(* CODESYS project CtaAppReport_3.0.0.0.library
   Description: Report Library der CTA
   Version: 3.0.0.0
   Title: CtaAppReport
   Author: SIS
   Company: CTA
   Placeholder: CtaAppReport
   DocFormat: reStructuredText
   CompiledLibraryCompatibilityVersion: CODESYS V3.5 SP16 Patch 3
   LanguageModelAttribute: qualified-access-only
   DefaultNamespace: CtaAppReport

Project tree, tasks and I/O mapping:
  libraries: Standard, 3.5.18.0 (System); CtaAppBmk, 2.0.0.0 (CTA); CtaSysConfig, 1.0.0.2 (CTA); CtaVisSymbols, 1.0.0.0 (CTA); CtaSysEvent, 1.0.0.0 (CTA); VisuDialogs, 3.5.16.20 (System); SysFile, 3.5.17.0 (System); SysDir, 3.5.17.0 (System); VisuSymbols, 4.5.0.0 (System); StringUtils, 3.5.18.0 (System); SysTypes2 Interfaces, * (System); TextListUtils, * (System); CtaAppInfluxLog, 1.0.0.1 (CTA); CtaAppTime, 1.0.0.1 (CTA); SysProcess Implementation, 3.5.17.0 (System); CmpErrors, 3.3.1.40 (System); VisuElemBase, * (System)
  40 Visualizations/
    visualisation REPORT_ID
    TABLE/
      visualisation VIS_REPORT_TABLE
      visualisation VIS_REPORT_TABLE_BASE
      DELETE/
        visualisation VIS_REPORT_DELETE
    PUSHLINE/
      visualisation VIS_REPORT_PUSH_LINE
      visualisation VIS_REPORT_PUSH_LINE_BASE
      visualisation VIS_REPORT_PUSH_LINE_QUERRY
    TABLE LINE/
      visualisation VIS_REPORT_TABLE_LINE_BASE
      visualisation VIS_REPORT_TABLE_LINE_QUERRY
      visualisation VIS_REPORT_TABLE_LINE
    REPORTMANAGER/
      visualisation VIS_REPORTMANAGER
      visualisation VIS_REPORTMANAGER_BASE
    HAND/
      visualisation VIS_REPORT_HAND
    ANZAHL REPORTS/
      visualisation VIS_ANZ_REPORTS_OVERALL
      Modul/
        visualisation VIS_ANZ_REPORTS_MODUL
        visualisation VIS_ANZ_REPORTS_MODUL_BASE
        visualisation VIS_ANZ_REPORTS_MODUL_QUERRY
  30 Program Organization Units/
    CSV/
      function block fbDataHandler [ST]: metWriteDtFrom, FB_INIT, FB_EXIT, actInitPath, proGetCountsOfReports, proExportIdStart, metExportId, metResetCycleCount, proExport, proIsRegistred, metStartDone, metPrepeareStop, proDenyStop, metCyclicCall, metWriteOnChange, metDeleteHistory, metAddObjForeWriteDtFrom, metAddObjForeWriteDtTo, metAddObjForeWriteOnChange
    OBJ/
      function block fbReportObjectFactory [ST]: metQuittAllReports, metDestroyCsvReportObject, metQuittSelectedReports, metCsvGetItf, metDestroyReportObject, metGetItf, metCreateReportObject, proGetNextPos, proGetAktiveReport, proGetActiveErrorMbString, proIsThereAnAktiveError, proGetActiveWarningMbString, metReSaveAfterDelete, metGarbageControll, GetActiveErrorModbusLanguageString
      function block fbReportObject [ST]: proGetReporterText, proGetReportText, proAdditionalText, proCountRetry, proIsQuitt, proIsSelected, proMaxRetry, proReportAcknowledgType, proReportId, proReportTextId, proReportTextList, proReportType, proReporterObjectId, proStateActive, proWritePosInCsv, proQuitt, metSendDataToInflux, metReportObject, proReportIn, proDtFrom, proDtTo, proSetMetaData, metDestroy, proPrio, metWriteDtFromToCsv, metWriteDtToToCsv, metSaveOnChange, metGarbage, GetReportTextLanguage
      function fcWordToHexString [ST]
      function fcReportIdToString8 [ST]
    REPORTER/
      function block fbReportManager [ST]: proWarningText, metSyncReporter, proInfoText, proErrorText, proGetErrorNr, actInit, proGetWarningNr, proGetInfoNr, proAnzError, proAnzWarning, proAnzInfo, proTotalReports
      function block fbReporter [ST]: metGetQuitt, proAktivReport, proHandLokal, proNewReport, metReport, proGetCounts, proDoneReport, proPrio, proOptionalText
    VIS/
      function block fbReportVisu [ST]: metGetReport, metGetShowReport, actConfigFile, proQuittExtern, loadHistory, actEWI, FB_INIT, metReload, FilterWarning, SetFilterId, loadPending, FilterInfo, FilterError, proAnzReportsInTable, proIdMissmatch, MaxOffset
    function fcBmkToId [ST]
    SORT/
      function block fbSort [ST]: metSortPrio, metFilterCustom, proAnzAktiveError, proAnzAktiveInfo, proAnzAktiveReports, proAnzAktiveWarning, proAnzReportsInTable
    program REPORT [ST]
    SQL/
      function Fc_MariaDbDeleteHistory [ST]
      function Fc_MariaDbLogWrite [ST]
      function Fc_MariaDbLogRead [ST]
      function Fc_MariaDbHighestId [ST]
  00000000-0000-0000-0000-000000000000|D:\CoDeSys\LibrariesV3\trunk\Intern\CAA\CAA Template\3.4.0.0 draft\Placeholder.xml
  00000000-0000-0000-0000-000000000000|D:\CoDeSys\LibrariesV3\trunk\Intern\CAA\CAA Template\3.2.0.3 draft\Prefix.pdf
  00000000-0000-0000-0000-000000000000|D:\CoDeSys\LibrariesV3\trunk\Intern\CAA\CAA Template\3.5.2.0 draft\Placeholder.xml
  20 Structs/
    data type enReportType
    data type scPara
    data type scReportMetaData
    data type scReportNr
    data type stReportTextList
    data type enReportacknowledgeType
    data type enTableType
    data type ST_MariaDbLog
  50 Images/
  10 Documenation/
    global variables VersionHistory
    global variables readMe
  21 Interface/
    interface ITF_REPORTMANAGER: proErrorText, proGetWarningNr, metSyncReporter, proGetErrorNr, proGetInfoNr, proInfoText, proWarningText, proTotalReports
    interface ITF_REPORTOBJECT: proGetReportText, proStateActive, proIsQuitt, proIsSelected, proReportId, proMaxRetry, proCountRetry, proReportTextList, proReportTextId, proReporterObjectId, proAdditionalText, proReportType, proReportAcknowledgType, proWritePosInCsv, proGetReporterText, proReportIn, proDtTo, proDtFrom, metReportObject, proQuitt, proSetMetaData, proPrio, metDestroy, metWriteDtFromToCsv, metSaveOnChange, GetReportTextLanguage
  11 Library Parameter/
    global variables Parameter
  12 Konstanten/
    global variables GlobalKonstant
  60 Textlisten/
    text list txtLibAp99_1Error
    text list txtLibAp99_2enTypeOfAck
    text list txtLibAp99_2Warnung
    text list txtLibAp99_3Info
    text list GlobalTextList
    text list txtNoTextList
  13 Globale Variablen/
    global variables GVL_Report
    global variables GVL_REPORT_PERSISTENT
*)

// 20 Structs/enReportType
TYPE enReportType :
(
	Info    := 0,
    Warning := 1,
    Error   := 2
);
END_TYPE

// 20 Structs/scPara
TYPE scPara :
    STRUCT
        fbxEnSafetyFernQuitt            :   CtaSysConfig.fbBOOL;
        fbuiMaxFernQuitt                :   CtaSysConfig.fbUINT;         
    END_STRUCT
END_TYPE

// 20 Structs/scReportMetaData
TYPE scReportMetaData :
    STRUCT
        xReportIn                   :   BOOL;                           // Report Input
        xActive                     :   BOOL;                           // State of Report
        xIsQuitt                    :   BOOL;                           // State of Acknowledge
        xQuitt                      :   BOOL;                           // Acknowledge Flag
        xIsSelected                 :   BOOL;                           // State of Selected in Table
        dtFrom                      :   DT;                             // Date and Time of Report happen
        dtTo                        :   DT;                             // Date and Time of Report gone
        iMaxRetry                   :   INT;                            // Max allowed Retries till Acknowledge is required
        iCountRetry                 :   INT;                            // Retries till now
        stReportTxtId               :   STRING[3];                      // Report Id fore Texlist
        stReportTextList            :   STRING[100];                    // Report TextList 
        uliReportId                 :   ULINT;                          // Report Id build out of BMK and Report Text Id. Ex: Bmk 56M111 & Id 3 = 567711103  
        enReportType                :   enReportType;                   // Type of Report
        enReportacknowledgeType     :   enReportacknowledgeType;        // Type of Report Acknowledge
        stReporterObjId             :   STRING[20];                     // Object Id of Reporter      
        stAdditionalText            :   STRING[20];                     // Additional Text
        dwWritePosInCsv             :   DWORD;                          // Position in Csv File fore write dtTo 
        usiPrio                     :   USINT;                          // Prio
    END_STRUCT
END_TYPE

// 20 Structs/scReportNr
TYPE scReportNr :
    STRUCT
        iError              :   INT;            // Error Status
        usiErrorPrio        :   USINT;
        iWarning            :   INT;            // Warning Status
        usiWarnungPrio      :   USINT;
        iInfo               :   INT;            // Info Status
        usiInfoPrio         :   USINT;
    END_STRUCT
END_TYPE

// 20 Structs/stReportTextList
TYPE stReportTextList : STRING[100]; END_TYPE

// 20 Structs/enReportacknowledgeType
TYPE enReportacknowledgeType :
(
	Auto        := 0,
    Quit        := 1,
    RetryN      := 2
);
END_TYPE

// 20 Structs/enTableType
{attribute 'qualified_only'}
{attribute 'strict'}
TYPE enTableType :
(
	PENDING_REPORTS := 0,
    HISTORY_REPORTS := 1
);
END_TYPE

// 20 Structs/ST_MariaDbLog
TYPE ST_MariaDbLog :
	STRUCT
		id                       : ULINT;
		createdAt                : DT;
		reportType               : enReportType;
		reportId                 : ULINT;
		reporterText             : STRING(150);
		reportText               : STRING(140);
		dtFrom                   : DT;
		dtTo                     : DT;
		isQuitt                  : BOOL;
		reportTextList           : STRING(100);
		reportTextId              : STRING(3);
		reportAcknowledgType     : USINT;
		objectId                 : STRING(20);
		instancePath             : STRING(255);
		additionalText           : STRING(20);
		prio                     : USINT;
		reportIn                  : BOOL;
		stateActive               : BOOL;
	END_STRUCT
END_TYPE

// 10 Documenation/VersionHistory
(* 

.. image:: ../../Images/CTA_Logo.jpg
   :align: right
   :width: 15% 

**Vorlage**   


============ =========== =========== ============================================
**Date**     **Version** **Author**  **Change**
------------ ----------- ----------- --------------------------------------------
04.03.2021   0.0.0.0     SIS         Vorlage erstellt

============ =========== =========== ============================================


*)
VAR_GLOBAL
    stInfo : STRING:= '0.0.0.0, Vorlage, CTA';
END_VAR

// 10 Documenation/readMe
(*

**ReadMe**
 
|	**Empfehlung**
|
|	Die LibAp99aErrorManagement wird benötigt damit aus dem BMK der CTA-E-Schema eine Störungsnummer generiert werden kann. 
|	Es wird für die Ausgabe ein DINT verwendet. Die aufschlüsselung von Buchstaben wird durch die ASCI Nr ersetzt.     
|  
| *Beispiel* 
|
| BMK             =   **56M11**    
| Fehler Nr       =   01-10
| ErrorNr-Modbus  =   BMK    + Fehler Nr
| 56771101        =   567711 + 01
| 56771102        =   567711 + 02
| 56771103        =   567711 + 03
| 56771104        =   567711 + 04
| 56771105        =   567711 + 05
| 56771106        =   567711 + 06
| 56771107        =   567711 + 07 
| 56771108        =   567711 + 08
| 56771109        =   567711 + 09
| 56771110        =   567711 + 10 
|
| Wenn der Fehler keiner BMK zugeordnet werden kann, sollte von der Nr. 1000 hochgezähl werden. 
| Tiefere Nr. werden von den Bibliotheken benötigt. 
*)

VAR_GLOBAL
    xReadMeDone              :   BOOL;
END_VAR

// 13 Globale Variablen/GVL_Report
{attribute 'qualified_only'}
VAR_GLOBAL
    fbReportObjectFactory     :   fbReportObjectFactory;
    fbSort                    :   fbSort;
    fbReportVisu              :   fbReportVisu;
    (* Reports *)             
    ayReportObject            :   ARRAY[1..Parameter.diMaxObject] OF fbReportObject;
    ayItfAktiveReports        :   ARRAY[1..Parameter.diMaxObject] OF ITF_REPORTOBJECT;
    ayItfSortetReportsPrio    :   ARRAY[1..Parameter.diMaxObject] OF ITF_REPORTOBJECT;
    ayItfSortetReportsCustom  :   ARRAY[0..GlobalKonstant.VISU_MAX_NUMBER_OF_CLIENTS] OF ARRAY[1..Parameter.diMaxObject] OF ITF_REPORTOBJECT;
    ayCsvReportObject         :   ARRAY[0..GlobalKonstant.VISU_MAX_NUMBER_OF_CLIENTS] OF ARRAY[0..GlobalKonstant.iUpperSizeTable] OF fbReportObject;
    fbDataHandler             :   fbDataHandler;
    diCountHand               :   DINT;
END_VAR

// 11 Library Parameter/Parameter
{attribute 'qualified_only'}
VAR_GLOBAL CONSTANT
    diMaxObject                  :   DINT :=  150;   // Max 200
    diMaxExportsPerCycle         :   DINT :=  50;    // Kann sich auf die Zykluszeit auswirken wenn zu viele Id pro Zyklus exportiert werden
END_VAR

// 12 Konstanten/GlobalKonstant
{attribute 'qualified_only'}
VAR_GLOBAL CONSTANT
    stTextListWarning           :   stReportTextList    := 'CtaAppReport.txtLibAp99_2Warnung';
    stTextListInfo              :   stReportTextList    := 'CtaAppReport.txtLibAp99_3Info';
    iUpperSizeTable             :   INT                 := 13;   
	VISU_MAX_NUMBER_OF_CLIENTS	:	INT					:= 15;
END_VAR

// 13 Globale Variablen/GVL_REPORT_PERSISTENT
{attribute 'qualified_only'}
VAR_GLOBAL RETAIN 
	scLastErrorReport         :   scReportMetaData;
	scLastWarningReport       :   scReportMetaData;
	scLastInfoReport          :   scReportMetaData;  
END_VAR

// 21 Interface/ITF_REPORTMANAGER
INTERFACE ITF_REPORTMANAGER EXTENDS __SYSTEM.IQueryInterface

PROPERTY proErrorText : STRING[100]
GET
END_GET
END_PROPERTY

PROPERTY proGetWarningNr : INT
GET
END_GET
END_PROPERTY

METHOD metSyncReporter : BOOL
VAR_INPUT
	refFbReporter	:	REFERENCE TO fbReporter;
END_VAR
END_METHOD

PROPERTY proGetErrorNr : INT
GET
END_GET
END_PROPERTY

PROPERTY proGetInfoNr : INT
GET
END_GET
END_PROPERTY

PROPERTY proInfoText : STRING[100]
GET
END_GET
END_PROPERTY

PROPERTY proWarningText : STRING[100]
GET
END_GET
END_PROPERTY

PROPERTY proTotalReports : INT
GET
END_GET
END_PROPERTY

END_INTERFACE

// 30 Program Organization Units/REPORTER/fbReporter
FUNCTION_BLOCK FINAL fbReporter 
VAR
	diArrayReportAdr     :	DINT;
	iCountReports		 :	INT;
	tonDelay			 :	TON;
	tonReset			 :	TON;
	_stReportTextList    :	POINTER TO stReportTextList;
	_iReportID			 :  INT;
	xNewReport			 :  BOOL;
	xAktiveReport		 :  BOOL;
    xDoneReport          :  BOOL;
	_enReportType        :  enReportType;
    xHand                :  BOOL;
    usiPrio              :  USINT;
    xExportDone          :  BOOL; 
    xInitDone            :  BOOL;
END_VAR

METHOD metGetQuitt : BOOL
VAR
    ITF_REPORTOBJECT : ITF_REPORTOBJECT;
END_VAR
IF diArrayReportAdr >= 1 THEN
    IF __QUERYINTERFACE(GVL_Report.fbReportObjectFactory.metGetItf(diArrayReportAdr),ITF_REPORTOBJECT) THEN
        metGetQuitt := ITF_REPORTOBJECT.proIsQuitt;
    END_IF;
ELSE
    metGetQuitt := FALSE;
END_IF
END_METHOD

PROPERTY proAktivReport : BOOL
GET
proAktivReport := xAktiveReport;
END_GET
END_PROPERTY

PROPERTY proHandLokal : BOOL
SET
IF proHandLokal AND  NOT xHand THEN
    GVL_Report.diCountHand := GVL_Report.diCountHand + 1;
    xHand := TRUE;
ELSIF NOT proHandLokal AND xHand THEN
    GVL_Report.diCountHand := GVL_Report.diCountHand - 1;
    IF GVL_Report.diCountHand < 0 THEN
        GVL_Report.diCountHand := 0;
	END_IF;
    xHand := FALSE;    
END_IF;
END_SET
END_PROPERTY

PROPERTY INTERNAL proNewReport : BOOL
SET
xNewReport := proNewReport;
END_SET
GET
proNewReport := xNewReport;
END_GET
END_PROPERTY

METHOD FINAL metReport : BOOL
VAR_INPUT
    xSetReportIn          		:   BOOL;
    iReportID           		:   INT;
    enReportTypeIn      		:   enReportType;
    enReportAcknowledgeTypeIn   :   enReportAcknowledgeType;
	tDelay              		:   TIME;  
	ITF_BMK_IN					:	CtaAppBmk.ITF_BMK;
	pstReportTextListIn 		:	POINTER TO stReportTextList;	 
	stOptionalReportText		:	STRING[20];	
    iRetryTilReportLock 		:   INT;                            
    xResetCount         		:   BOOL;                            
	tReset						:	TIME;                 
END_VAR
VAR
    ITF_REPORTOBJECT            :   ITF_REPORTOBJECT;
END_VAR
IF xInitDone AND_THEN pstReportTextListIn <> 0 AND_THEN ITF_BMK_IN <> 0 THEN
    // Counter mit xResetCount rücksetzen wenn Count < iMaxRetry
    IF tReset > T#0MS AND_THEN enReportAcknowledgeTypeIn = enReportacknowledgeType.RetryN AND_THEN NOT xSetReportIn THEN
        tonReset.IN := iCountReports < iRetryTilReportLock AND iCountReports > 0;
        tonReset.PT	:= tReset;
        tonReset();
	ELSE
		tonReset(IN := FALSE,
				 PT := T#0MS);
    END_IF;
    IF (xResetCount OR tonReset.Q) AND_THEN iCountReports < iRetryTilReportLock AND NOT xSetReportIn  THEN
        diArrayReportAdr := 0;   
        iCountReports := 0;
        tonReset.IN := FALSE;
        tonReset.PT	:= T#0S;	 
        tonReset();
    END_IF;        
	IF xSetReportIn THEN	
		_stReportTextList    := pstReportTextListIn;	
		_iReportID 			 := iReportID;
		_enReportType		 := enReportTypeIn;
	END_IF;
	
	tonDelay.IN          := xSetReportIn;
	tonDelay.PT          := tDelay;
	tonDelay();
	(* Wenn Report nicht registriert Registrierprozess starten *)
    IF diArrayReportAdr = 0 THEN
        // Wenn tonDelay.Q aktiv Registrieren      
        IF tonDelay.Q THEN
            (* Create Report Object *)
            diArrayReportAdr := GVL_Report.fbReportObjectFactory.metCreateReportObject();   
            IF diArrayReportAdr <> 0 THEN 
                IF __QUERYINTERFACE(GVL_Report.fbReportObjectFactory.metGetItf(diArrayReportAdr),ITF_REPORTOBJECT) THEN               
                    (* Set Infos *)  
                    xNewReport := TRUE;
                    xAktiveReport := TRUE;
                    iCountReports := iCountReports + 1;
                    ITF_REPORTOBJECT.proReportType              :=  enReportTypeIn;                         // Report Type
                    ITF_REPORTOBJECT.proReportAcknowledgType    :=  enReportAcknowledgeTypeIn;              // Report Acknowledge Type
                    ITF_REPORTOBJECT.proReportTextId            :=  TO_STRING(iReportID);                   // Report Id
                    ITF_REPORTOBJECT.proReportTextList          :=  pstReportTextListIn^;                   // Report Text list
                    ITF_REPORTOBJECT.proReporterObjectId        :=  ITF_BMK_IN.proGetObjectId;              // Reporter Object Id
                    ITF_REPORTOBJECT.proSetInstancePath         :=  ITF_BMK_IN.proGetInstancePath;          // Reporter Instance Path
                    ITF_REPORTOBJECT.proMaxRetry                :=  iRetryTilReportLock;                    // Max Retries
                    ITF_REPORTOBJECT.proCountRetry              :=  iCountReports;                          // Countet Retries
                    ITF_REPORTOBJECT.proAdditionalText          :=  stOptionalReportText;                   // Additional Text
                    ITF_REPORTOBJECT.proReportIn                :=  xSetReportIn;                           // Report Input
                    ITF_REPORTOBJECT.proPrio                    :=  usiPrio;
                    ITF_REPORTOBJECT.metReportObject();                                                     // Call Object              
                END_IF                                                                 
            END_IF;
        END_IF;
    ELSE
        // Zyklische aktualisierung der Daten nach Registrierung       
        IF __QUERYINTERFACE(GVL_Report.fbReportObjectFactory.metGetItf(diArrayReportAdr),ITF_REPORTOBJECT) THEN
            IF ITF_REPORTOBJECT.proReportIn <> xSetReportIn THEN
                ITF_REPORTOBJECT.proReportIn :=  xSetReportIn;                                   // Report Input
            END_IF;
			// Nach Manuellem Quittieren Counts rücksetzen     
			IF ITF_REPORTOBJECT.proQuitt THEN
				iCountReports := 0;
			END_IF;              
			IF NOT ITF_REPORTOBJECT.proStateActive THEN
                xAktiveReport   := FALSE;   
                xDoneReport     := TRUE;
 
                diArrayReportAdr := 0;  
            END_IF;
            ITF_REPORTOBJECT.metReportObject();                                                             // Call Object 
        ELSE
            diArrayReportAdr := 0;
            xAktiveReport   := FALSE; 
            xDoneReport     := TRUE;
        END_IF;                                              
    END_IF;

    // ID Liste erzeugen
    IF GVL_Report.fbDataHandler.proExport AND NOT xExportDone THEN
        xExportDone :=  GVL_Report.fbDataHandler.metExportId(  ITF_BMK_IN	            := 	ITF_BMK_IN,
                                                              iID                       :=  iReportID,
                                                              enReportTypeIn            :=  enReportTypeIn,
                                                              enReportAcknowledgeTypeIn :=  enReportAcknowledgeTypeIn,
                                                              stReportTextListIn        :=  pstReportTextListIn^);
    ELSIF NOT GVL_Report.fbDataHandler.proExport THEN 
        xExportDone := FALSE;
    END_IF;  
END_IF;
xInitDone := TRUE;
END_METHOD

PROPERTY proGetCounts : INT
GET
proGetCounts := iCountReports;
END_GET
END_PROPERTY

PROPERTY proDoneReport : BOOL
SET
xDoneReport     := proDoneReport;
END_SET
GET
proDoneReport := xDoneReport;
END_GET
END_PROPERTY

PROPERTY proPrio : USINT
SET
IF proPrio <> usiPrio THEN
	usiPrio := proPrio;
END_IF;
END_SET
GET
proPrio := usiPrio;
END_GET
END_PROPERTY

PROPERTY proOptionalText : STRING(20)
GET
VAR
	ITF_REPORTOBJECT : ITF_REPORTOBJECT;
END_VAR
IF diArrayReportAdr <> 0 THEN
	IF __QUERYINTERFACE(GVL_Report.fbReportObjectFactory.metGetItf(diArrayReportAdr),ITF_REPORTOBJECT) THEN 
		proOptionalText := 	ITF_REPORTOBJECT.proAdditionalText;
	END_IF;
END_IF;
END_GET
END_PROPERTY

END_FUNCTION_BLOCK

// 30 Program Organization Units/OBJ/fbReportObjectFactory
FUNCTION_BLOCK fbReportObjectFactory
VAR_INPUT
END_VAR
VAR_OUTPUT
END_VAR
VAR 
    diNextFreePosition            :   DINT := 1;
	dwSync						  :   DWORD;
	old_language				  :   STRING(4)	:= 'oldL';
END_VAR

METHOD metQuittAllReports : BOOL
VAR
    diFor    :   DINT;
END_VAR
FOR diFor := 1 TO Parameter.diMaxObject DO
    IF GVL_Report.ayItfAktiveReports[diFor] <> 0 THEN
        IF GVL_Report.ayItfAktiveReports[diFor].proStateActive AND_THEN NOT GVL_Report.ayItfAktiveReports[diFor].proIsQuitt THEN
            GVL_Report.ayItfAktiveReports[diFor].proQuitt := TRUE;    
		END_IF;
	END_IF;
END_FOR;
END_METHOD

(* Destroy Report Object *)
METHOD PRIVATE metDestroyCsvReportObject : BOOL
VAR_INPUT
    iArrayPos   :   INT;
	diClientId		 :	 DINT;
END_VAR
IF iArrayPos >= 0 AND iArrayPos <= 9 THEN
    GVL_Report.ayCsvReportObject[diClientId][iArrayPos].metDestroy();
    metDestroyCsvReportObject := TRUE;
END_IF;
END_METHOD

METHOD metQuittSelectedReports : BOOL
VAR
    diFor    :   DINT;
END_VAR
FOR diFor := 1 TO Parameter.diMaxObject DO
    IF GVL_Report.ayItfAktiveReports[diFor] <> 0 THEN
        IF GVL_Report.ayItfAktiveReports[diFor].proIsSelected AND_THEN GVL_Report.ayItfAktiveReports[diFor].proStateActive AND_THEN NOT GVL_Report.ayItfAktiveReports[diFor].proIsQuitt THEN
            GVL_Report.ayItfAktiveReports[diFor].proQuitt := TRUE;    
		END_IF;
	END_IF;
END_FOR;
END_METHOD

METHOD metCsvGetItf : ITF_REPORTOBJECT
VAR_INPUT
    diArrayPos   :   DINT;
	diClientId	 :	 DINT;
END_VAR
IF diArrayPos >= 0 AND diArrayPos <= GlobalKonstant.iUpperSizeTable THEN    
    metCsvGetItf := GVL_Report.ayCsvReportObject[diClientId][diArrayPos];
END_IF;
END_METHOD

(* Destroy Report Object *)
METHOD PRIVATE metDestroyReportObject : BOOL
VAR_INPUT
    diArrayPos   :   DINT;
END_VAR
IF diArrayPos >= 1 AND diArrayPos <= Parameter.diMaxObject THEN   
    IF NOT GVL_Report.ayReportObject[diArrayPos].proStateActive THEN
        GVL_Report.ayReportObject[diArrayPos].metDestroy();
        metDestroyReportObject := TRUE;
    ELSE
        metDestroyReportObject := FALSE;
    END_IF;
END_IF;
END_METHOD

METHOD metGetItf : ITF_REPORTOBJECT
VAR_INPUT
    diArrayPos   :   DINT;
END_VAR
IF diArrayPos >= 1 AND diArrayPos <= Parameter.diMaxObject THEN
    metGetItf := GVL_Report.ayReportObject[diArrayPos];
END_IF;
END_METHOD

(* Returns Arrayposition of Object*) 
METHOD metCreateReportObject : DINT
VAR
    diCurrentPositon    :   DINT;
    diCurrentOverFlows  :   DINT;
    diSavetyCount       :   DINT;
	dwExklusiveAcces	:	DWORD;
END_VAR
REPEAT 
    metCreateReportObject := 0;
	dwExklusiveAcces := TEST_AND_SET(dwSync);
	IF dwExklusiveAcces = 0 THEN
		IF diNextFreePosition + 1 > Parameter.diMaxObject THEN
			diCurrentPositon    := __XADD(ADR(diNextFreePosition),-Parameter.diMaxObject + 1);
		ELSE
			diCurrentPositon := __XADD(ADR(diNextFreePosition),1);  
		END_IF;
		dwSync := 0;
	END_IF;
    IF diCurrentPositon >= 1 AND diCurrentPositon <= Parameter.diMaxObject THEN
        IF NOT GVL_Report.ayReportObject[diCurrentPositon].proStateActive THEN
            metDestroyReportObject(diCurrentPositon);
            metCreateReportObject := diCurrentPositon;     
            metDestroyReportObject(diNextFreePosition);
        END_IF;
    END_IF;
    diSavetyCount := diSavetyCount + 1;
UNTIL
    metCreateReportObject <> 0 OR diSavetyCount >= Parameter.diMaxObject
END_REPEAT;
END_METHOD

PROPERTY proGetNextPos : DINT
GET
proGetNextPos := diNextFreePosition;
END_GET
END_PROPERTY

PROPERTY proGetAktiveReport : ITF_REPORTOBJECT
GET
proGetAktiveReport := GVL_Report.ayItfSortetReportsPrio[1];
END_GET
END_PROPERTY

PROPERTY proGetActiveErrorMbString : STRING(160)
GET
VAR
    ITF_REPORTOBJECT_TEMP   :   ITF_REPORTOBJECT;
END_VAR
(* Error Nr as String *)
proGetActiveErrorMbString := '';
IF __QUERYINTERFACE(proGetAktiveReport,ITF_REPORTOBJECT_TEMP) THEN
    IF ITF_REPORTOBJECT_TEMP.proReportType = enReportType.Error THEN
        proGetActiveErrorMbString := CONCAT(fcReportIdToString8(ITF_REPORTOBJECT_TEMP.proReportId),CONCAT(' ',CONCAT(ITF_REPORTOBJECT_TEMP.proGetBMK,CONCAT(' ',ITF_REPORTOBJECT_TEMP.proGetReportText))));       
    ELSE
        RETURN;
	END_IF;
END_IF;
END_GET
END_PROPERTY

PROPERTY proIsThereAnAktiveError : BOOL
GET
VAR
    diFor   :   DINT;
END_VAR
proIsThereAnAktiveError := FALSE;
FOR diFor := 1 TO Parameter.diMaxObject DO
    IF GVL_Report.ayItfSortetReportsPrio[diFor] <> 0 THEN
        IF GVL_Report.ayItfSortetReportsPrio[diFor].proStateActive THEN
            IF GVL_Report.ayItfSortetReportsPrio[diFor].proReportType = enReportType.Error THEN
                proIsThereAnAktiveError := TRUE;
                EXIT;    
            ELSE
                CONTINUE;
            END_IF;
        ELSE
            CONTINUE;
        END_IF;
    ELSE
        CONTINUE;
    END_IF;
END_FOR;
END_GET
END_PROPERTY

PROPERTY proGetActiveWarningMbString : STRING(160)
GET
VAR
    ITF_REPORTOBJECT_TEMP   :   ITF_REPORTOBJECT;
    diFor                   :   DINT;
END_VAR
(* Error Nr as String *)
proGetActiveWarningMbString := '';
// Warning
FOR diFor := Parameter.diMaxObject TO 1 BY -1 DO 
    IF GVL_Report.ayItfSortetReportsPrio[diFor] <> 0 AND_THEN GVL_Report.ayItfSortetReportsPrio[diFor].proStateActive AND_THEN GVL_Report.ayItfSortetReportsPrio[diFor].proReportType = enReportType.Warning THEN
        ITF_REPORTOBJECT_TEMP :=  GVL_Report.ayItfSortetReportsPrio[diFor];   
        RETURN;
    END_IF;        
END_FOR;
IF ITF_REPORTOBJECT_TEMP <> 0 THEN
        proGetActiveWarningMbString := CONCAT(fcReportIdToString8(ITF_REPORTOBJECT_TEMP.proReportId),CONCAT(' ',CONCAT(ITF_REPORTOBJECT_TEMP.proGetBMK,CONCAT(' ',ITF_REPORTOBJECT_TEMP.proGetReportText))));       
END_IF;
END_GET
END_PROPERTY

METHOD metReSaveAfterDelete : BOOL
VAR
    diFor    :   DINT;
END_VAR
FOR diFor := 1 TO Parameter.diMaxObject DO
    IF GVL_Report.ayItfAktiveReports[diFor] <> 0 THEN
        GVL_Report.ayItfAktiveReports[diFor].metWriteDtFromToCsv(); 
	END_IF;
END_FOR;
END_METHOD

METHOD metGarbageControll : BOOL
VAR
    diFor   :   DINT;
END_VAR
metGarbageControll := FALSE;   
FOR diFor := 1 TO Parameter.diMaxObject DO
    IF GVL_Report.ayReportObject[diFor].proStateActive THEN
        IF GVL_Report.ayReportObject[diFor].metGarbage() THEN     
        	metGarbageControll := TRUE;   
		END_IF;
	END_IF;
END_FOR;
END_METHOD

METHOD GetActiveErrorModbusLanguageString : STRING(160)
VAR_INPUT
	language	:	STRING(4);
END_VAR
VAR
    ITF_REPORTOBJECT_TEMP   :   ITF_REPORTOBJECT;
END_VAR
(* Error Nr as String *)
GetActiveErrorModbusLanguageString := '';
IF __QUERYINTERFACE(proGetAktiveReport,ITF_REPORTOBJECT_TEMP) THEN
    IF ITF_REPORTOBJECT_TEMP.proReportType = enReportType.Error THEN
		IF old_language <> language THEN
			CmpDynamicText.DynamicTextLoadLanguage(language);
			old_language := language;
		END_IF;
        GetActiveErrorModbusLanguageString := CONCAT(fcReportIdToString8(ITF_REPORTOBJECT_TEMP.proReportId),CONCAT(' ',CONCAT(ITF_REPORTOBJECT_TEMP.proGetBMK,CONCAT(' ',ITF_REPORTOBJECT_TEMP.GetReportTextLanguage(language)))));       
    ELSE
        RETURN;
	END_IF;
END_IF;
END_METHOD

END_FUNCTION_BLOCK

// 30 Program Organization Units/REPORT
PROGRAM REPORT
VAR
END_VAR

(* Csv Fb *)
GVL_Report.fbDataHandler();
(* Visu Fb *)
GVL_Report.fbReportVisu();
(* Prüfen ob Objecte Unbrauchbar sind *)
IF GVL_Report.fbReportObjectFactory.metGarbageControll() THEN
	(* Tabelle neu Laden wenn Objecte zerstört *)
    GVL_Report.fbSort.metSortPrio();
END_IF;

END_PROGRAM

// 30 Program Organization Units/CSV/fbDataHandler
FUNCTION_BLOCK fbDataHandler IMPLEMENTS CtaSysEvent.ITF_APPEVENT
VAR CONSTANT
    wSize               :   WORD    :=  786;  
    wSizeHeader         :   WORD    :=  150;
END_VAR
VAR
	stFilePathHistory   :   STRING;
    stFileDownloadHtml  :   STRING;
    stFilePathDelete    :   STRING;
    xInitDone           :   BOOL;
    xIsNotSimulation    :   BOOL;
    stSpace             :   STRING[1] := ' ';
    stRN                :   STRING[1] := '$R';
    stSC                :   STRING[1] := ';';
    stHeader            :   STRING[wSizeHeader]; 
    stHtmlDownload      :   STRING[88];
    RTS_IEC_RESULT_Ini  :   RTS_IEC_RESULT;
    RTS_IEC_HANDLE_Ini  :   RTS_IEC_HANDLE;     
    RTS_IEC_RESULT_Exp  :   RTS_IEC_RESULT;
    RTS_IEC_HANDLE_ExE  :   RTS_IEC_HANDLE; 
    RTS_IEC_HANDLE_ExW  :   RTS_IEC_HANDLE;    
    RTS_IEC_HANDLE_ExI  :   RTS_IEC_HANDLE;   
    FILE_STATUS         :   SysFile.SYS_FILE_STATUS; 
    xExportId           :   BOOL;
    xExportPossible     :   BOOL;
    xIsExporting        :   BOOL;
    xExportDoneTemp     :   BOOL;
    xExportDone         :   BOOL;
    dwWrite             :   DWORD;
    diCountExp          :   DINT;
    iWait               :   INT;
    xIsRegistretAppEvent:   BOOL;
    ITF_BMK_NEXT_EXPORT :   CtaAppBmk.ITF_BMK;

	dwSync				:	DWORD;
	ayITF_WriteDtFrom	:	ARRAY[0..Parameter.diMaxObject] OF ITF_REPORTOBJECT;
	diNextFreeDtFrom	:	DINT;
	diNextFreeDtFromOld	:	DINT;
	ayITF_WriteDtTo		:	ARRAY[0..Parameter.diMaxObject] OF ITF_REPORTOBJECT;
	diNextFreeDtTo		:	DINT;
	diNextFreeDtToOld	:	DINT;
	ayITF_WriteChange	:	ARRAY[0..Parameter.diMaxObject] OF ITF_REPORTOBJECT;
	diNextFreeChange	:	DINT;
	diNextFreeChangeOld	:	DINT;
	diFor				:	DINT;
	udiCurrentMaxIndex	:	UDINT;
END_VAR;

(* Dt From *)
IF diNextFreeDtFrom <> diNextFreeDtFromOld THEN
	FOR diFor := LOWER_BOUND(ayITF_WriteDtFrom,1) TO UPPER_BOUND(ayITF_WriteDtFrom,1) DO
		IF ayITF_WriteDtFrom[diFor] <> 0 THEN
			metWriteDtFrom(ayITF_WriteDtFrom[diFor]);
			ayITF_WriteDtFrom[diFor] := 0;
		END_IF;
	END_FOR;
	diNextFreeDtFromOld := diNextFreeDtFrom;
ELSE
	diNextFreeDtFrom 	:= 0;
	diNextFreeDtFromOld	:= 0;
END_IF;

(* Change *)
IF diNextFreeChange <> diNextFreeChangeOld THEN
	FOR diFor := LOWER_BOUND(ayITF_WriteChange,1) TO UPPER_BOUND(ayITF_WriteChange,1) DO
		IF ayITF_WriteChange[diFor] <> 0 THEN
			metWriteOnChange(ayITF_WriteChange[diFor]);
			ayITF_WriteChange[diFor] := 0;
		END_IF;
	END_FOR;
	diNextFreeChangeOld := diNextFreeChange;
ELSE
	diNextFreeChange 	:= 0;
	diNextFreeChangeOld	:= 0;	
END_IF;

(* DtTo *)
IF diNextFreeDtTo <> diNextFreeDtToOld THEN
	FOR diFor := LOWER_BOUND(ayITF_WriteDtTo,1) TO UPPER_BOUND(ayITF_WriteDtTo,1)  DO
		IF ayITF_WriteDtTo[diFor] <> 0 THEN
			metWriteOnChange(ayITF_WriteDtTo[diFor]);
			ayITF_WriteDtTo[diFor] := 0;
		END_IF;
	END_FOR;
	diNextFreeDtToOld := diNextFreeDtTo;
ELSE
	diNextFreeDtTo 		:= 0;
	diNextFreeDtToOld	:= 0;	
END_IF;

METHOD PRIVATE metWriteDtFrom : DWORD
VAR_INPUT
    ITF_REPORTOBJECT_IN : ITF_REPORTOBJECT;
END_VAR
VAR
    ITF_REPORTOBJECT_QUERY  :   ITF_REPORTOBJECT;
	dwResultTemp	:	DWORD;
END_VAR
IF __QUERYINTERFACE(ITF_REPORTOBJECT_IN,ITF_REPORTOBJECT_QUERY) THEN
	
   Fc_MariaDbLogWrite(	xExecute				:= TRUE, 
					update_id				:= ITF_REPORTOBJECT_QUERY.proWritePosInCsv, 
					proReportType			:= ITF_REPORTOBJECT_QUERY.proReportType, 
					proReportId				:= ITF_REPORTOBJECT_QUERY.proReportId, 
					proGetReporterText		:= ITF_REPORTOBJECT_QUERY.proGetReporterText, 
					proGetReportText		:= ITF_REPORTOBJECT_QUERY.proGetReportText, 
					proDtFrom				:= ITF_REPORTOBJECT_QUERY.proDtFrom, 
					proDtTo					:= ITF_REPORTOBJECT_QUERY.proDtTo, 
					proIsQuitt				:= ITF_REPORTOBJECT_QUERY.proIsQuitt, 
					proReportTextList		:= ITF_REPORTOBJECT_QUERY.proReportTextList, 
					proReportTextId			:= ITF_REPORTOBJECT_QUERY.proReportTextId, 
					proReportAcknowledgType	:= TO_USINT(ITF_REPORTOBJECT_QUERY.proReportAcknowledgType), 
					proGetObjectId			:= ITF_REPORTOBJECT_QUERY.proGetObjectId, 
					proGetInstancePath		:= ITF_REPORTOBJECT_QUERY.proGetInstancePath, 
					proAdditionalText		:= ITF_REPORTOBJECT_QUERY.proAdditionalText, 
					proPrio					:= ITF_REPORTOBJECT_QUERY.proPrio, 
					proReportIn				:= ITF_REPORTOBJECT_QUERY.proReportIn, 
					proStateActive			:= ITF_REPORTOBJECT_QUERY.proStateActive,
					dwResult				=> dwResultTemp);
					udiCurrentMaxIndex := MAX(udiCurrentMaxIndex,TO_UDINT(dwResultTemp));
					ITF_REPORTOBJECT_QUERY.proWritePosInCsv := dwResultTemp;
					
   
END_IF;
END_METHOD

//FB_Init ist immer implizit verfügbar und wird primär für die Initialisierung verwendet.
//Der Rückgabewert wird nicht ausgewertet. Für gezielte Einflussnahme können Sie
//die Methoden explizit deklarieren und darin mit dem Standard-Initialisierungscode 
//zusätzlichen Code bereitstellen. Sie können den Rückgabewert auswerten.
METHOD FB_Init: BOOL
VAR_INPUT    
bInitRetains: BOOL; // TRUE: Die Retain-Variablen werden initialisiert (Reset warm / Reset kalt)    
bInCopyCode: BOOL;  // TRUE: Die Instanz wird danach in den Kopiercode kopiert (Online-Change)
END_VAR
actInitPath();
CtaSysEvent.fcRegistry(THIS^);
END_METHOD

//FB_Exit muss explizit implementiert werden. Wenn es eine Implementierung gibt, dann wird 
//die Methode aufgerufen, bevor die Steuerung den Code der Funktionsbaustein-Instanz entfernt
//(impliziter Aufruf. Der Rückgabewert wird nicht ausgewertet.
METHOD FB_Exit: BOOL
VAR_INPUT    
bInCopyCode: BOOL;  // TRUE: Die Exit-Methode wird aufgerufen, um die Instanz zu verlassen, die hinterher kopiert wird Online-Change).  
END_VAR
END_METHOD

ACTION actInitPath:
IF NOT xInitDone THEN
	__TRY
    {IF NOT defined (IsSimulationMode)}
                    
        xIsNotSimulation := TRUE;                                                     
    {END_IF}   
	
    // Download Html erzeugen
    IF xIsNotSimulation THEN
        (* ID-Download *)    
            stFileDownloadHtml  :=  '';
            stFileDownloadHtml  :=  './visu/History/IDDownload.htm';                
            RTS_IEC_HANDLE_Ini := SysFile.SysFileOpen(stFileDownloadHtml,SysFile.ACCESS_MODE.AM_WRITE_PLUS,ADR(RTS_IEC_RESULT_Ini));
            // Schreibe Position festlegen
            SysFile.SysFileSetPos(RTS_IEC_HANDLE_Ini,0); 
            stHtmlDownload  := '';      
            stHtmlDownload  := '<HTML><HEAD><TITLE></TITLE></HEAD><BODY>';
            // Daten Schreiben
            SysFile.SysFileWrite(RTS_IEC_HANDLE_Ini,ADR(stHtmlDownload),TO_DWORD(LEN(stHtmlDownload)),ADR(RTS_IEC_RESULT_Ini));           
            stHtmlDownload  := '';      
            stHtmlDownload  := '<a href="Export/E_ID.csv" download = "E_ID.csv">E-ID Download</a><br />';                                                     
            // Daten Schreiben
            SysFile.SysFileWrite(RTS_IEC_HANDLE_Ini,ADR(stHtmlDownload),TO_DWORD(LEN(stHtmlDownload)),ADR(RTS_IEC_RESULT_Ini)); 
            stHtmlDownload  := '';      
            stHtmlDownload  := '<a href="Export/W_ID.csv" download = "W_ID.csv">W-ID Download</a><br />';                                                     
            // Daten Schreiben
            SysFile.SysFileWrite(RTS_IEC_HANDLE_Ini,ADR(stHtmlDownload),TO_DWORD(LEN(stHtmlDownload)),ADR(RTS_IEC_RESULT_Ini));                                                        
            stHtmlDownload  := '';      
            stHtmlDownload  := '<a href="Export/I_ID.csv" download = "I_ID.csv">I-ID Download</a><br />';                                                     
            // Daten Schreiben
            SysFile.SysFileWrite(RTS_IEC_HANDLE_Ini,ADR(stHtmlDownload),TO_DWORD(LEN(stHtmlDownload)),ADR(RTS_IEC_RESULT_Ini));                 
            stHtmlDownload  := '';      
            stHtmlDownload  := '</BODY></HTML>';                                                     
            // Daten Schreiben
            SysFile.SysFileWrite(RTS_IEC_HANDLE_Ini,ADR(stHtmlDownload),TO_DWORD(LEN(stHtmlDownload)),ADR(RTS_IEC_RESULT_Ini));                                                 
            SysFile.SysFileClose(RTS_IEC_HANDLE_Ini);                  
           RTS_IEC_HANDLE_Ini := 0;
            stFileDownloadHtml  :=  '';
            stFileDownloadHtml  :=  'History/HistoryDownload.htm';
        END_IF;        

    IF xIsNotSimulation THEN
            stFilePathDelete := '';
            stFilePathDelete := './visu/History/Export/E_ID.csv';
            SysFile.SysFileDelete(stFilePathDelete);
            stFilePathDelete := '';
            stFilePathDelete := './visu/History/Export/W_ID.csv';
            SysFile.SysFileDelete(stFilePathDelete);
            stFilePathDelete := '';            
            stFilePathDelete := './visu/History/Export/I_ID.csv';    
            SysFile.SysFileDelete(stFilePathDelete);        
    ELSE
            stFilePathDelete := '';
            stFilePathDelete := 'C:/PFC_Simulation/visu/History/Export/E_ID.csv';
            SysFile.SysFileDelete(stFilePathDelete);
            stFilePathDelete := '';
            stFilePathDelete := 'C:/PFC_Simulation/visu/History/Export/W_ID.csv';
            SysFile.SysFileDelete(stFilePathDelete);
            stFilePathDelete := '';
            stFilePathDelete := 'C:/PFC_Simulation/visu/History/Export/I_ID.csv';  
            SysFile.SysFileDelete(stFilePathDelete);
    END_IF;  
	Fc_MariaDbDeleteHistory(xExecute := TRUE,dwResult => udiCurrentMaxIndex);
    xInitDone := TRUE;
	__CATCH
		xInitDone := TRUE;
	__ENDTRY
END_IF;
END_ACTION

PROPERTY proGetCountsOfReports : UDINT
GET
proGetCountsOfReports := udiCurrentMaxIndex;
END_GET
END_PROPERTY

PROPERTY proExportIdStart : BOOL
SET
VAR
    stTemp  :   STRING(255);
END_VAR
IF proExportIdStart AND NOT xExportId THEN
    xExportId := TRUE;
    stTemp    := '';
    stTemp    := './visu/History/Export/E_ID.csv';
    RTS_IEC_HANDLE_ExE := SysFile.SysFileOpen(stTemp,ACCESS_MODE.AM_WRITE_PLUS,ADR(RTS_IEC_RESULT_Exp));
    stTemp    := '';
    stTemp    := './visu/History/Export/W_ID.csv';
    RTS_IEC_HANDLE_ExW := SysFile.SysFileOpen(stTemp,ACCESS_MODE.AM_WRITE_PLUS,ADR(RTS_IEC_RESULT_Exp));
    stTemp    := '';
    stTemp    := './visu/History/Export/I_ID.csv';
    RTS_IEC_HANDLE_ExI := SysFile.SysFileOpen(stTemp,ACCESS_MODE.AM_WRITE_PLUS,ADR(RTS_IEC_RESULT_Exp));    
    stTemp    := '';
    stTemp    := 'REPORT TYPE;ID;BMK;AKS;VENDOR DESIGNATION;REPORT TEXT$R';
    SysFile.SysFileWrite(RTS_IEC_HANDLE_ExE,ADR(stTemp),TO_UINT(LEN(stTemp)),ADR(RTS_IEC_RESULT_Exp));    
    SysFile.SysFileWrite(RTS_IEC_HANDLE_ExW,ADR(stTemp),TO_UINT(LEN(stTemp)),ADR(RTS_IEC_RESULT_Exp));
    SysFile.SysFileWrite(RTS_IEC_HANDLE_ExI,ADR(stTemp),TO_UINT(LEN(stTemp)),ADR(RTS_IEC_RESULT_Exp));   
END_IF
END_SET
GET
proExportIdStart := xExportId;
END_GET
END_PROPERTY

METHOD metExportId : BOOL
VAR_INPUT
    ITF_BMK_IN                  :   CtaAppBmk.ITF_BMK;
    stReportTextListIn          :   stReportTextList;
    iId                         :   INT;
    enReportTypeIn      		:   enReportType;
    enReportAcknowledgeTypeIn   :   enReportAcknowledgeType;    
END_VAR
VAR
    stTemp                      :   STRING(255);
    stId                        :   STRING(3);
    ITF_BMK_QUERY               :   CtaAppBmk.ITF_BMK;     
    RTS_IEC_HANDLE_Exp          :   RTS_IEC_HANDLE;
    diIndex                     :   DINT;
END_VAR
IF ITF_BMK_NEXT_EXPORT = ITF_BMK_IN THEN
    ITF_BMK_NEXT_EXPORT := 0;
    diIndex :=__XADD(ADR(diCountExp),-diCountExp);
END_IF;
diIndex :=__XADD(ADR(diCountExp),1);
IF diIndex <= Parameter.diMaxExportsPerCycle THEN
    xIsExporting := TRUE;
    (* Type of Report *)
    stTemp := '';
    IF enReportTypeIn = enReportType.Error THEN
        stTemp := 'ERROR';
        RTS_IEC_HANDLE_Exp  := RTS_IEC_HANDLE_ExE;
    ELSIF enReportTypeIn = enReportType.Warning THEN
        stTemp := 'WARNING';
        RTS_IEC_HANDLE_Exp  := RTS_IEC_HANDLE_ExW;
    ELSIF enReportTypeIn = enReportType.Info THEN   
        stTemp := 'INFO';
        RTS_IEC_HANDLE_Exp  := RTS_IEC_HANDLE_ExI;
    END_IF;
    (* Check Handle *)    
    IF RTS_IEC_HANDLE_Exp <> 0 AND __QUERYINTERFACE(ITF_BMK_IN,ITF_BMK_QUERY) THEN
        (* Write Type *)
        SysFile.SysFileWrite(RTS_IEC_HANDLE_Exp,ADR(stTemp),TO_UINT(LEN(stTemp)),ADR(RTS_IEC_RESULT_Exp));
        (* Write Semicolon *)
        stTemp := '';
        stTemp := ';';
        SysFile.SysFileWrite(RTS_IEC_HANDLE_Exp,ADR(stTemp),TO_UINT(LEN(stTemp)),ADR(RTS_IEC_RESULT_Exp));
        (* Write ID *)
        stTemp := '';
        stTemp := TO_STRING(fcBmkToId(ITF_BMK_QUERY.proGetBMK,TO_DINT(iId),FALSE,enReportTypeIn));
        SysFile.SysFileWrite(RTS_IEC_HANDLE_Exp,ADR(stTemp),TO_UINT(LEN(stTemp)),ADR(RTS_IEC_RESULT_Exp));
        (* Write Semicolon *)
        stTemp := '';
        stTemp := ';';
        SysFile.SysFileWrite(RTS_IEC_HANDLE_Exp,ADR(stTemp),TO_UINT(LEN(stTemp)),ADR(RTS_IEC_RESULT_Exp));
        (* Write BMK *)
        stTemp := '';
        stTemp := ITF_BMK_QUERY.proGetBMK;
        SysFile.SysFileWrite(RTS_IEC_HANDLE_Exp,ADR(stTemp),TO_UINT(LEN(stTemp)),ADR(RTS_IEC_RESULT_Exp));
        (* Write Semicolon *)
        stTemp := '';
        stTemp := ';';
        SysFile.SysFileWrite(RTS_IEC_HANDLE_Exp,ADR(stTemp),TO_UINT(LEN(stTemp)),ADR(RTS_IEC_RESULT_Exp));    
        (* Write AKS *)
        stTemp := '';
        stTemp := ITF_BMK_QUERY.proGetAKS;
        SysFile.SysFileWrite(RTS_IEC_HANDLE_Exp,ADR(stTemp),TO_UINT(LEN(stTemp)),ADR(RTS_IEC_RESULT_Exp));
        (* Write Semicolon *)
        stTemp := '';
        stTemp := ';';
        SysFile.SysFileWrite(RTS_IEC_HANDLE_Exp,ADR(stTemp),TO_UINT(LEN(stTemp)),ADR(RTS_IEC_RESULT_Exp));        
        (* Write Vendordesignation*)
        stTemp := '';
        stTemp := ITF_BMK_QUERY.proGetVendorDesignation;
        IF stTemp = '' THEN
            stTemp := ITF_BMK_QUERY.proGetInstancePath;
		END_IF;
        SysFile.SysFileWrite(RTS_IEC_HANDLE_Exp,ADR(stTemp),TO_UINT(LEN(stTemp)),ADR(RTS_IEC_RESULT_Exp));
        (* Write Semicolon *)
        stTemp := '';
        stTemp := ';';
        SysFile.SysFileWrite(RTS_IEC_HANDLE_Exp,ADR(stTemp),TO_UINT(LEN(stTemp)),ADR(RTS_IEC_RESULT_Exp));    
        (* Write Report Text *)
        stTemp := '';
        (*Load Text By Language*)
        stId   := TO_STRING(iId);
        stTemp := CmpDynamicText.DynamicTextGetText(ADR(stReportTextListIn),ADR(stId))^;
        (* Load Default Text if no spezifig Language*)
        IF stTemp = '' THEN
            stTemp := CmpDynamicText.DynamicTextGetDefaultText(ADR(stReportTextListIn),ADR(stId))^;
        END_IF;
        SysFile.SysFileWrite(RTS_IEC_HANDLE_Exp,ADR(stTemp),TO_UINT(LEN(stTemp)),ADR(RTS_IEC_RESULT_Exp));
        (* Write $R *)
        stTemp := '';
        stTemp := '$R';
        SysFile.SysFileWrite(RTS_IEC_HANDLE_Exp,ADR(stTemp),TO_UINT(LEN(stTemp)),ADR(RTS_IEC_RESULT_Exp));        
        metExportId := TRUE;     
    END_IF;
ELSE
    IF ITF_BMK_NEXT_EXPORT = 0 THEN
        ITF_BMK_NEXT_EXPORT := ITF_BMK_IN;
    END_IF;    
END_IF;
END_METHOD

METHOD metResetCycleCount : BOOL
VAR_INPUT
END_VAR
IF xExportDoneTemp THEN
    iWait := iWait + 1;
END_IF;
IF xExportDoneTemp AND NOT xIsExporting AND iWait >= 10000 THEN
    xExportDone         := TRUE;
    xExportDoneTemp     := FALSE;
    xExportId           := FALSE;
    ITF_BMK_NEXT_EXPORT := 0;
    diCountExp          := 0;
    IF RTS_IEC_HANDLE_ExE <> 0 THEN
        SysFile.SysFileClose(RTS_IEC_HANDLE_ExE);
        RTS_IEC_HANDLE_ExE  := 0;
    END_IF;
    IF RTS_IEC_HANDLE_ExW <> 0 THEN
        SysFile.SysFileClose(RTS_IEC_HANDLE_ExW);
        RTS_IEC_HANDLE_ExW  := 0;
    END_IF;
    IF RTS_IEC_HANDLE_ExI <> 0 THEN
        SysFile.SysFileClose(RTS_IEC_HANDLE_ExI);
        RTS_IEC_HANDLE_ExI  := 0;
    END_IF;    
END_IF;
IF xIsExporting THEN
    xExportDoneTemp := TRUE;
    xExportDone     := FALSE;
    xIsExporting    := FALSE;
    iWait           := 0;
END_IF;
END_METHOD

PROPERTY proExport : BOOL
GET
proExport := xExportId;
END_GET
END_PROPERTY

PROPERTY proIsRegistred : BOOL
SET
xIsRegistretAppEvent := proIsRegistred;
END_SET
GET
proIsRegistred := xIsRegistretAppEvent;
END_GET
END_PROPERTY

METHOD metStartDone : BOOL
RETURN;
END_METHOD

METHOD metPrepeareStop : BOOL
END_METHOD

PROPERTY proDenyStop : BOOL
GET
proDenyStop := NOT xInitDone;
END_GET
END_PROPERTY

METHOD metCyclicCall : BOOL
(* Reset CycleCount Csv *)
metResetCycleCount();
END_METHOD

METHOD PRIVATE metWriteOnChange : BOOL
VAR_INPUT
    ITF_REPORTOBJECT_IN 	: ITF_REPORTOBJECT;
END_VAR
VAR
    ITF_REPORTOBJECT_QUERY  :   ITF_REPORTOBJECT;
	dwResultTemp			:	DWORD;
END_VAR
IF __QUERYINTERFACE(ITF_REPORTOBJECT_IN,ITF_REPORTOBJECT_QUERY) THEN
	
   Fc_MariaDbLogWrite(	xExecute				:= TRUE, 
					update_id				:= ITF_REPORTOBJECT_QUERY.proWritePosInCsv, 
					proReportType			:= ITF_REPORTOBJECT_QUERY.proReportType, 
					proReportId				:= ITF_REPORTOBJECT_QUERY.proReportId, 
					proGetReporterText		:= ITF_REPORTOBJECT_QUERY.proGetReporterText, 
					proGetReportText		:= ITF_REPORTOBJECT_QUERY.proGetReportText, 
					proDtFrom				:= ITF_REPORTOBJECT_QUERY.proDtFrom, 
					proDtTo					:= ITF_REPORTOBJECT_QUERY.proDtTo, 
					proIsQuitt				:= ITF_REPORTOBJECT_QUERY.proIsQuitt, 
					proReportTextList		:= ITF_REPORTOBJECT_QUERY.proReportTextList, 
					proReportTextId			:= ITF_REPORTOBJECT_QUERY.proReportTextId, 
					proReportAcknowledgType	:= TO_USINT(ITF_REPORTOBJECT_QUERY.proReportAcknowledgType), 
					proGetObjectId			:= ITF_REPORTOBJECT_QUERY.proGetObjectId, 
					proGetInstancePath		:= ITF_REPORTOBJECT_QUERY.proGetInstancePath, 
					proAdditionalText		:= ITF_REPORTOBJECT_QUERY.proAdditionalText, 
					proPrio					:= ITF_REPORTOBJECT_QUERY.proPrio, 
					proReportIn				:= ITF_REPORTOBJECT_QUERY.proReportIn, 
					proStateActive			:= ITF_REPORTOBJECT_QUERY.proStateActive,
					dwResult				=> dwResultTemp);
					ITF_REPORTOBJECT_QUERY.proWritePosInCsv := dwResultTemp;
   
END_IF;
END_METHOD

METHOD metDeleteHistory : BOOL
VAR_INPUT
END_VAR
VAR
	diForTemp		:	DINT;
	temp_interface	:	ITF_REPORTOBJECT;
END_VAR
Fc_MariaDbDeleteHistory(xExecute := TRUE);
udiCurrentMaxIndex := 0;
FOR diForTemp := LOWER_BOUND(GVL_Report.ayItfAktiveReports,1) TO UPPER_BOUND(GVL_Report.ayItfAktiveReports,1) DO
	IF __QUERYINTERFACE(GVL_Report.ayItfAktiveReports[diForTemp],temp_interface) THEN
		GVL_Report.ayItfAktiveReports[diForTemp].proWritePosInCsv := 0;
		metAddObjForeWriteDtFrom(GVL_Report.ayItfAktiveReports[diForTemp]);
		IF GVL_Report.ayItfAktiveReports[diForTemp].proDtTo > TO_DT(0) THEN
			metAddObjForeWriteDtTo(GVL_Report.ayItfAktiveReports[diForTemp]);
		END_IF
	END_IF
END_FOR
GVL_Report.fbReportVisu.metReload();
END_METHOD

METHOD metAddObjForeWriteDtFrom
VAR_INPUT
	ITF_REPORTOBJECT_IN 	: ITF_REPORTOBJECT;	
END_VAR
VAR
	diOldValue				: DINT;
END_VAR
IF __QUERYINTERFACE(ITF_REPORTOBJECT_IN,ITF_REPORTOBJECT_IN) THEN
		diOldValue	:= __XADD(ADR(diNextFreeDtFrom),1);	
		IF diOldValue >= LOWER_BOUND(ayITF_WriteDtFrom,1) AND diOldValue <= UPPER_BOUND(ayITF_WriteDtFrom,1) THEN
			ayITF_WriteDtFrom[diOldValue] := ITF_REPORTOBJECT_IN;
		END_IF;
END_IF;
END_METHOD

METHOD metAddObjForeWriteDtTo
VAR_INPUT
	ITF_REPORTOBJECT_IN 	: ITF_REPORTOBJECT;	
END_VAR
VAR
	diOldValue				: DINT;
END_VAR
IF __QUERYINTERFACE(ITF_REPORTOBJECT_IN,ITF_REPORTOBJECT_IN) THEN
	IF ITF_REPORTOBJECT_IN.proWritePosInCsv > 0 THEN
		diOldValue	:= __XADD(ADR(diNextFreeDtTo),1);	
		IF diOldValue >= LOWER_BOUND(ayITF_WriteDtTo,1) AND diOldValue <= UPPER_BOUND(ayITF_WriteDtTo,1) THEN
			ayITF_WriteDtTo[diOldValue] := ITF_REPORTOBJECT_IN;
		END_IF;
	END_IF;
END_IF;
END_METHOD

METHOD metAddObjForeWriteOnChange
VAR_INPUT
	ITF_REPORTOBJECT_IN 	: ITF_REPORTOBJECT;	
END_VAR
VAR
	diOldValue				: DINT;
END_VAR
IF __QUERYINTERFACE(ITF_REPORTOBJECT_IN,ITF_REPORTOBJECT_IN) THEN
	IF ITF_REPORTOBJECT_IN.proWritePosInCsv > 0 THEN
		diOldValue	:= __XADD(ADR(diNextFreeChange),1);	
		IF diOldValue >= LOWER_BOUND(ayITF_WriteChange,1) AND diOldValue <= UPPER_BOUND(ayITF_WriteChange,1) THEN
			ayITF_WriteChange[diOldValue] := ITF_REPORTOBJECT_IN;
		END_IF;
	END_IF;	
END_IF;
END_METHOD

END_FUNCTION_BLOCK

// 21 Interface/ITF_REPORTOBJECT
INTERFACE ITF_REPORTOBJECT EXTENDS CtaAppBmk.ITF_BMK;

PROPERTY FINAL proGetReportText : STRING[140]
GET
END_GET
END_PROPERTY

PROPERTY FINAL proStateActive : BOOL
SET
END_SET
GET
END_GET
END_PROPERTY

PROPERTY FINAL proIsQuitt : BOOL
SET
END_SET
GET
END_GET
END_PROPERTY

PROPERTY FINAL proIsSelected : BOOL
SET
END_SET
GET
END_GET
END_PROPERTY

PROPERTY FINAL proReportId : ULINT
GET
END_GET
END_PROPERTY

PROPERTY FINAL proMaxRetry : INT
SET
END_SET
GET
END_GET
END_PROPERTY

PROPERTY FINAL proCountRetry : INT
SET
END_SET
GET
END_GET
END_PROPERTY

PROPERTY FINAL proReportTextList : STRING[100]
SET
END_SET
GET
END_GET
END_PROPERTY

PROPERTY FINAL proReportTextId : STRING[3]
SET
END_SET
GET
END_GET
END_PROPERTY

PROPERTY FINAL proReporterObjectId : STRING[20]
SET
END_SET
GET
END_GET
END_PROPERTY

PROPERTY FINAL proAdditionalText : STRING(20)
SET
END_SET
GET
END_GET
END_PROPERTY

PROPERTY FINAL proReportType : enReportType
SET
END_SET
GET
END_GET
END_PROPERTY

PROPERTY FINAL proReportAcknowledgType : enReportacknowledgeType
SET
END_SET
GET
END_GET
END_PROPERTY

PROPERTY FINAL proWritePosInCsv : DWORD
SET
END_SET
GET
END_GET
END_PROPERTY

PROPERTY FINAL proGetReporterText : STRING[150]
GET
END_GET
END_PROPERTY

PROPERTY FINAL proReportIn : BOOL
SET
END_SET
GET
END_GET
END_PROPERTY

PROPERTY FINAL proDtTo : DT
SET
END_SET
GET
END_GET
END_PROPERTY

PROPERTY FINAL proDtFrom : DT
SET
END_SET
GET
END_GET
END_PROPERTY

METHOD FINAL metReportObject : BOOL
VAR_INPUT
END_VAR
END_METHOD

PROPERTY FINAL proQuitt : BOOL
SET
END_SET
GET
END_GET
END_PROPERTY

PROPERTY FINAL proSetMetaData : scReportMetaData
SET
END_SET
END_PROPERTY

PROPERTY FINAL proPrio : USINT
SET
END_SET
GET
END_GET
END_PROPERTY

METHOD FINAL metDestroy
VAR_INPUT
END_VAR
END_METHOD

METHOD FINAL metWriteDtFromToCsv : DWORD
VAR_INPUT
END_VAR
END_METHOD

METHOD FINAL metSaveOnChange : BOOL
VAR_INPUT
END_VAR
END_METHOD

METHOD GetReportTextLanguage : STRING[140]
VAR_INPUT
	language	:	STRING(4);
END_VAR
END_METHOD

END_INTERFACE

// 30 Program Organization Units/SQL/Fc_MariaDbLogWrite
FUNCTION Fc_MariaDbLogWrite
VAR_INPUT
    xExecute 			   : BOOL;
	update_id			   : DWORD;
    proReportType          : enReportType;
    proReportId            : ULINT;
    proGetReporterText     : STRING(150);
    proGetReportText       : STRING(140);
    proDtFrom              : DT;
    proDtTo                : DT;
    proIsQuitt             : BOOL;
    proReportTextList      : STRING(100);
    proReportTextId        : STRING(3);
    proReportAcknowledgType: USINT;
    proGetObjectId         : STRING(20);
    proGetInstancePath     : STRING(255);
    proAdditionalText      : STRING(20);
    proPrio                : USINT;
    proReportIn            : BOOL;
    proStateActive         : BOOL;
END_VAR

VAR_OUTPUT
    xBusy       : BOOL;
    xDone       : BOOL;
    xError      : BOOL;
    dwResult    : DWORD;
END_VAR

VAR
    sCommand    : STRING(4095);
    sSQL        : STRING(4095);
    sStdOut     : STRING(1024);	
	sFind		: STRING := 'LAST_INSERT_ID()$N';
    xExecuteOld : BOOL;

    sType       : STRING(20);

    sObjectName : STRING(150);
    sReportText : STRING(140);
    sTextList   : STRING(100);
    sObjectId   : STRING(20);
    sInstance   : STRING(255);
    sAddText    : STRING(20);

    sDtFrom     : STRING(40);
    sDtTo       : STRING(40);

	sTemp		: STRING(1024);
    Result      : RTS_IEC_RESULT;

    diStdOutLen : DINT;
END_VAR

// Ausgänge zurücksetzen
xDone := FALSE;
xError := FALSE;
xBusy := TRUE;
dwResult := 0;
sStdOut := '';
sType 	:= '';
sTemp	:= '';
sCommand:= '';
// =====================================================
// REPORT TYPE
// =====================================================

IF proReportType = enReportType.Error THEN
	sType := 'ERROR';

ELSIF proReportType = enReportType.Warning THEN
	sType := 'WARNING';

ELSIF proReportType = enReportType.Info THEN
	sType := 'INFO';

ELSE
	sType := 'UNKNOWN';
END_IF;


// =====================================================
// DATEN IN STRINGS UMWANDELN
// =====================================================

sObjectName := proGetReporterText;

sReportText := proGetReportText;

sTextList := proReportTextList;

sObjectId := proGetObjectId;

sInstance := proGetInstancePath;

sAddText := proAdditionalText;


// =====================================================
// DATUM
// =====================================================

sDtFrom := TO_STRING(proDtFrom);
sDtFrom := DELETE(sDtFrom,3,1);
sDtTo := TO_STRING(proDtTo);
sDtTo := DELETE(sDtTo,3,1);

// =====================================================
// SQL AUFBAUEN
// =====================================================
IF update_id > 0 THEN
	sSQL 	:= '';
	sTemp	:=  'UPDATE logs SET ';
	StrConcatA(ADR(sTemp),ADR(sSQL),TO_INT(SIZEOF(sSQL)));			
ELSE
	sSQL 	:= '';
	sTemp	:=  'INSERT INTO logs SET ';
	StrConcatA(ADR(sTemp),ADR(sSQL),TO_INT(SIZEOF(sSQL)));		
END_IF;

// -----------------------------------------------------
// event_title
// -----------------------------------------------------
sTemp 	:= '';
sTemp	:= 'event_title = $'';
StrConcatA(ADR(sTemp),ADR(sSQL),TO_INT(SIZEOF(sSQL)));

sTemp 	:= '';
sTemp	:= sType;
StrConcatA(ADR(sTemp),ADR(sSQL),TO_INT(SIZEOF(sSQL)));

sTemp 	:= '';
sTemp	:= ' ';
StrConcatA(ADR(sTemp),ADR(sSQL),TO_INT(SIZEOF(sSQL)));

sTemp 	:= '';
sTemp	:= proGetReporterText;
StrConcatA(ADR(sTemp),ADR(sSQL),TO_INT(SIZEOF(sSQL)));

sTemp 	:= '';
sTemp	:= ' ';
StrConcatA(ADR(sTemp),ADR(sSQL),TO_INT(SIZEOF(sSQL)));

sTemp 	:= '';
sTemp	:= proGetReportText;
StrConcatA(ADR(sTemp),ADR(sSQL),TO_INT(SIZEOF(sSQL)));

sTemp 	:= '';
sTemp	:= '$',';
StrConcatA(ADR(sTemp),ADR(sSQL),TO_INT(SIZEOF(sSQL)));	

// -----------------------------------------------------
// event_type
// -----------------------------------------------------
sTemp 	:= '';
sTemp	:= 'event_type = $'';
StrConcatA(ADR(sTemp),ADR(sSQL),TO_INT(SIZEOF(sSQL)));

sTemp 	:= '';
sTemp	:= sType;
StrConcatA(ADR(sTemp),ADR(sSQL),TO_INT(SIZEOF(sSQL)));

sTemp 	:= '';
sTemp	:= '$',';
StrConcatA(ADR(sTemp),ADR(sSQL),TO_INT(SIZEOF(sSQL)));	

// -----------------------------------------------------
// event_id
// -----------------------------------------------------
sTemp 	:= '';
sTemp	:= 'event_id = ';
StrConcatA(ADR(sTemp),ADR(sSQL),TO_INT(SIZEOF(sSQL)));

sTemp 	:= '';
sTemp	:= ULINT_TO_STRING(proReportId);
StrConcatA(ADR(sTemp),ADR(sSQL),TO_INT(SIZEOF(sSQL)));

sTemp 	:= '';
sTemp	:= ',';
StrConcatA(ADR(sTemp),ADR(sSQL),TO_INT(SIZEOF(sSQL)));

// -----------------------------------------------------
// object_name
// -----------------------------------------------------
sTemp 	:= '';
sTemp	:= 'object_name = $'';
StrConcatA(ADR(sTemp),ADR(sSQL),TO_INT(SIZEOF(sSQL)));

sTemp 	:= '';
sTemp	:= sObjectName;
StrConcatA(ADR(sTemp),ADR(sSQL),TO_INT(SIZEOF(sSQL)));

sTemp 	:= '';
sTemp	:= '$',';
StrConcatA(ADR(sTemp),ADR(sSQL),TO_INT(SIZEOF(sSQL)));	

// -----------------------------------------------------
// reporttext
// -----------------------------------------------------
sTemp 	:= '';
sTemp	:= 'reporttext = $'';
StrConcatA(ADR(sTemp),ADR(sSQL),TO_INT(SIZEOF(sSQL)));

sTemp 	:= '';
sTemp	:= sReportText;
StrConcatA(ADR(sTemp),ADR(sSQL),TO_INT(SIZEOF(sSQL)));

sTemp 	:= '';
sTemp	:= '$',';
StrConcatA(ADR(sTemp),ADR(sSQL),TO_INT(SIZEOF(sSQL)));	

// -----------------------------------------------------
// dt_from
// -----------------------------------------------------
sTemp 	:= '';
sTemp	:= 'dt_from = $'';
StrConcatA(ADR(sTemp),ADR(sSQL),TO_INT(SIZEOF(sSQL)));

sTemp 	:= '';
sTemp	:= sDtFrom;
StrConcatA(ADR(sTemp),ADR(sSQL),TO_INT(SIZEOF(sSQL)));

sTemp 	:= '';
sTemp	:= '$',';
StrConcatA(ADR(sTemp),ADR(sSQL),TO_INT(SIZEOF(sSQL)));	

// -----------------------------------------------------
// dt_to
// -----------------------------------------------------
sTemp 	:= '';
sTemp	:= 'dt_to = $'';
StrConcatA(ADR(sTemp),ADR(sSQL),TO_INT(SIZEOF(sSQL)));

sTemp 	:= '';
sTemp	:= sDtTo;
StrConcatA(ADR(sTemp),ADR(sSQL),TO_INT(SIZEOF(sSQL)));

sTemp 	:= '';
sTemp	:= '$',';
StrConcatA(ADR(sTemp),ADR(sSQL),TO_INT(SIZEOF(sSQL)));	

// -----------------------------------------------------
// is_quitt
// -----------------------------------------------------

IF proIsQuitt THEN
	sTemp 	:= '';
	sTemp	:= 'is_quitt = TRUE,';
	StrConcatA(ADR(sTemp),ADR(sSQL),TO_INT(SIZEOF(sSQL)));
ELSE
	sTemp 	:= '';
	sTemp	:= 'is_quitt = FALSE,';
	StrConcatA(ADR(sTemp),ADR(sSQL),TO_INT(SIZEOF(sSQL)));
END_IF;

// -----------------------------------------------------
// report_textlist
// -----------------------------------------------------
sTemp 	:= '';
sTemp	:= 'report_textlist = $'';
StrConcatA(ADR(sTemp),ADR(sSQL),TO_INT(SIZEOF(sSQL)));

sTemp 	:= '';
sTemp	:= sTextList;
StrConcatA(ADR(sTemp),ADR(sSQL),TO_INT(SIZEOF(sSQL)));

sTemp 	:= '';
sTemp	:= '$',';
StrConcatA(ADR(sTemp),ADR(sSQL),TO_INT(SIZEOF(sSQL)));	

// -----------------------------------------------------
// text_id
// -----------------------------------------------------
sTemp 	:= '';
sTemp	:= 'text_id = ';
StrConcatA(ADR(sTemp),ADR(sSQL),TO_INT(SIZEOF(sSQL)));

sTemp 	:= '';
sTemp	:= proReportTextId;
StrConcatA(ADR(sTemp),ADR(sSQL),TO_INT(SIZEOF(sSQL)));

sTemp 	:= '';
sTemp	:= ',';
StrConcatA(ADR(sTemp),ADR(sSQL),TO_INT(SIZEOF(sSQL)));

// -----------------------------------------------------
// acknowledgement type
// -----------------------------------------------------
sTemp 	:= '';
sTemp	:= 'type_acknowledg = ';
StrConcatA(ADR(sTemp),ADR(sSQL),TO_INT(SIZEOF(sSQL)));

sTemp 	:= '';
sTemp	:= USINT_TO_STRING(proReportAcknowledgType);
StrConcatA(ADR(sTemp),ADR(sSQL),TO_INT(SIZEOF(sSQL)));

sTemp 	:= '';
sTemp	:= ',';
StrConcatA(ADR(sTemp),ADR(sSQL),TO_INT(SIZEOF(sSQL)));

// -----------------------------------------------------
// object_id
// -----------------------------------------------------
sTemp 	:= '';
sTemp	:= 'object_id = $'';
StrConcatA(ADR(sTemp),ADR(sSQL),TO_INT(SIZEOF(sSQL)));

sTemp 	:= '';
sTemp	:= sObjectId;
StrConcatA(ADR(sTemp),ADR(sSQL),TO_INT(SIZEOF(sSQL)));

sTemp 	:= '';
sTemp	:= '$',';
StrConcatA(ADR(sTemp),ADR(sSQL),TO_INT(SIZEOF(sSQL)));	

// -----------------------------------------------------
// instance_path
// -----------------------------------------------------
sTemp 	:= '';
sTemp	:= 'instance_path = $'';
StrConcatA(ADR(sTemp),ADR(sSQL),TO_INT(SIZEOF(sSQL)));

sTemp 	:= '';
sTemp	:= sInstance;
StrConcatA(ADR(sTemp),ADR(sSQL),TO_INT(SIZEOF(sSQL)));

sTemp 	:= '';
sTemp	:= '$',';
StrConcatA(ADR(sTemp),ADR(sSQL),TO_INT(SIZEOF(sSQL)));	

// -----------------------------------------------------
// additional_text
// -----------------------------------------------------
sTemp 	:= '';
sTemp	:= 'additional_text = $'';
StrConcatA(ADR(sTemp),ADR(sSQL),TO_INT(SIZEOF(sSQL)));

sTemp 	:= '';
sTemp	:= sAddText;
StrConcatA(ADR(sTemp),ADR(sSQL),TO_INT(SIZEOF(sSQL)));

sTemp 	:= '';
sTemp	:= '$',';
StrConcatA(ADR(sTemp),ADR(sSQL),TO_INT(SIZEOF(sSQL)));	

// -----------------------------------------------------
// priority
// -----------------------------------------------------
sTemp 	:= '';
sTemp	:= 'prio = ';
StrConcatA(ADR(sTemp),ADR(sSQL),TO_INT(SIZEOF(sSQL)));	

sTemp 	:= '';
sTemp	:= USINT_TO_STRING(proPrio);
StrConcatA(ADR(sTemp),ADR(sSQL),TO_INT(SIZEOF(sSQL)));

sTemp 	:= '';
sTemp	:= ',';
StrConcatA(ADR(sTemp),ADR(sSQL),TO_INT(SIZEOF(sSQL)));

// -----------------------------------------------------
// IN
// -----------------------------------------------------
IF proReportIn THEN
	sTemp 	:= '';
	sTemp	:= 'in_state = TRUE,';
	StrConcatA(ADR(sTemp),ADR(sSQL),TO_INT(SIZEOF(sSQL)));
ELSE
	sTemp 	:= '';
	sTemp	:= 'in_state = FALSE,';
	StrConcatA(ADR(sTemp),ADR(sSQL),TO_INT(SIZEOF(sSQL)));
END_IF;

// -----------------------------------------------------
// STATE
// -----------------------------------------------------
IF proStateActive THEN
	IF update_id > 0 THEN
		sTemp 	:= '';
		sTemp	:= 'state = TRUE';
		StrConcatA(ADR(sTemp),ADR(sSQL),TO_INT(SIZEOF(sSQL)));		

		sTemp 	:= '';
		sTemp	:= ' WHERE id = ';
		StrConcatA(ADR(sTemp),ADR(sSQL),TO_INT(SIZEOF(sSQL)));	
		 
		sTemp 	:= '';
		sTemp	:= UDINT_TO_STRING(DWORD_TO_UDINT(update_id));
		StrConcatA(ADR(sTemp),ADR(sSQL),TO_INT(SIZEOF(sSQL)));	
		
		sTemp 	:= '';
		sTemp	:= ';';
		StrConcatA(ADR(sTemp),ADR(sSQL),TO_INT(SIZEOF(sSQL)));				
	ELSE
		sTemp 	:= '';
		sTemp	:= 'state = TRUE;';
		StrConcatA(ADR(sTemp),ADR(sSQL),TO_INT(SIZEOF(sSQL)));		
	END_IF
ELSE
	IF update_id > 0 THEN
		sTemp 	:= '';
		sTemp	:= 'state = FALSE';
		StrConcatA(ADR(sTemp),ADR(sSQL),TO_INT(SIZEOF(sSQL)));		

		sTemp 	:= '';
		sTemp	:= ' WHERE id = ';
		StrConcatA(ADR(sTemp),ADR(sSQL),TO_INT(SIZEOF(sSQL)));	
		 
		sTemp 	:= '';
		sTemp	:= UDINT_TO_STRING(DWORD_TO_UDINT(update_id));
		StrConcatA(ADR(sTemp),ADR(sSQL),TO_INT(SIZEOF(sSQL)));	
		
		sTemp 	:= '';
		sTemp	:= ';';
		StrConcatA(ADR(sTemp),ADR(sSQL),TO_INT(SIZEOF(sSQL)));				
	ELSE
		sTemp 	:= '';
		sTemp	:= 'state = FALSE;';
		StrConcatA(ADR(sTemp),ADR(sSQL),TO_INT(SIZEOF(sSQL)));		
	END_IF
END_IF;

// =====================================================
// LINUX COMMAND
// =====================================================
sCommand := '';
sTemp := '';
sTemp := 'mariadb --socket=/var/lib/mysql/mysql.sock -u root -pCTA-MariaDb1981! --default-character-set=utf8mb4 -e "';
StrConcatA(ADR(sTemp),ADR(sCommand),TO_INT(SIZEOF(sCommand)));

sTemp := '';
sTemp := 'CREATE DATABASE IF NOT EXISTS CtaMariaDb; ';
StrConcatA(ADR(sTemp),ADR(sCommand),TO_INT(SIZEOF(sCommand)));

sTemp := '';
sTemp := 'USE CtaMariaDb;
CREATE TABLE IF NOT EXISTS logs (
	id BIGINT UNSIGNED AUTO_INCREMENT PRIMARY KEY,
	created_at DATETIME NOT NULL DEFAULT CURRENT_TIMESTAMP,
	event_title TEXT,
	event_type VARCHAR(20) NOT NULL,
	event_id BIGINT NOT NULL,
	object_name VARCHAR(255),
	reporttext TEXT,
	dt_from DATETIME NULL,
	dt_to DATETIME NULL,
	is_quitt BOOLEAN,
	report_textlist VARCHAR(255),
	text_id INT,
	type_acknowledg INT,
	object_id VARCHAR(50),
	instance_path VARCHAR(500),
	additional_text TEXT,
	prio INT,
	in_state BOOLEAN,
	state BOOLEAN,
	INDEX idx_dt_from (dt_from),
	INDEX idx_event_id (event_id),
	INDEX idx_object_id (object_id)
);';
StrConcatA(ADR(sTemp),ADR(sCommand),TO_INT(SIZEOF(sCommand)));	

StrConcatA(ADR(sSQL),ADR(sCommand),TO_INT(SIZEOF(sCommand)));	

sTemp := '';
sTemp := ' SELECT LAST_INSERT_ID();"';
StrConcatA(ADR(sTemp),ADR(sCommand),TO_INT(SIZEOF(sCommand)));

// =====================================================
// SYSPROCESS
// =====================================================

diStdOutLen :=
	SysProcess_Implementation.SysProcessExecuteCommand2(
		pszCommand := sCommand,
		pszStdOut := sStdOut,
		udiStdOutLen := SIZEOF(sStdOut),
		pResult := ADR(Result)
	);
IF update_id = 0 THEN
	IF Stu.StrFindA(ADR(sStdOut),ADR(sFind),0) > 0 THEN
		Stu.StrDeleteA(ADR(sStdOut),Stu.LEN(sFind),1);
		dwResult := TO_DWORD(sStdOut);
	ELSE
		dwResult := 0;
	END_IF;
ELSE
	dwResult := update_id;
END_IF;

// =====================================================
// ERGEBNIS
// =====================================================

IF Result = CmpErrors.Errors.ERR_OK THEN

	xDone := TRUE;
	xError := FALSE;

ELSE

	xDone := FALSE;
	xError := TRUE;

END_IF;

xBusy := FALSE;

END_FUNCTION

// 30 Program Organization Units/SQL/Fc_MariaDbDeleteHistory
FUNCTION Fc_MariaDbDeleteHistory
VAR_INPUT
    xExecute 			   : BOOL;
END_VAR

VAR_OUTPUT
    xBusy       : BOOL;
    xDone       : BOOL;
    xError      : BOOL;
    dwResult    : DWORD;
END_VAR

VAR
    sCommand    : STRING(1024);
    sStdOut     : STRING(100);	
	sFind		: STRING := 'MAX(id)$N';
    xExecuteOld : BOOL;

	sTemp		: STRING(1024);
    Result      : RTS_IEC_RESULT;

    diStdOutLen : DINT;
END_VAR

// Ausgänge zurücksetzen
xDone := FALSE;
xError := FALSE;
xBusy := TRUE;
dwResult := 0;
sStdOut := '';
sTemp	:= '';
sCommand:= '';

// =====================================================
// LINUX COMMAND
// =====================================================
sCommand := '';
sTemp := '';
sTemp := 'mariadb --socket=/var/lib/mysql/mysql.sock -u root -pCTA-MariaDb1981! --default-character-set=utf8mb4 CtaMariaDb -e "TRUNCATE TABLE logs;"';
StrConcatA(ADR(sTemp),ADR(sCommand),TO_INT(SIZEOF(sCommand)));

// =====================================================
// SYSPROCESS
// =====================================================

diStdOutLen :=
	SysProcess_Implementation.SysProcessExecuteCommand2(
		pszCommand := sCommand,
		pszStdOut := sStdOut,
		udiStdOutLen := SIZEOF(sStdOut),
		pResult := ADR(Result)
	);

// =====================================================
// ERGEBNIS
// =====================================================

IF Result = CmpErrors.Errors.ERR_OK THEN

	xDone := TRUE;
	xError := FALSE;

ELSE

	xDone := FALSE;
	xError := TRUE;

END_IF;

xBusy := FALSE;

END_FUNCTION

// 30 Program Organization Units/fcBmkToId
FUNCTION fcBmkToId  :   ULINT;
VAR_INPUT
    stBMK           :   STRING             [8];                                                                     // BMK als STRING [8]
    diNr            :   DINT;                                                                                       // Nr welche am ende angefügt wird
    xNoZero         :   BOOL;                                                                                       // Bei 1-Stelliger Nummer keine 0 voransetzen
    enReportTypeIn  :   enReportType;
END_VAR
VAR
    iFor            :   INT;                                                                                        // Forschleifen Variable
    iOfset          :   INT;                                                                                        // Offsetvariable 
    pstBMK          :   POINTER TO STRING  [8];                                                                    // Pointer auf stBMK
    pstBmkAscii     :   POINTER TO STRING  [12];                                                                    // Pointer auf stBmkAscii
    stBmkAscii      :   STRING             [12];                                                                    // String mit dem Numerischen BMK Code
    iAkt            :   INT;
END_VAR

//===========================================================================================================================================================================================================================================//
//  Pointer zuweisung		                                                                          																															             //
//===========================================================================================================================================================================================================================================// 
pstBMK          := ADR(stBMK);
pstBmkAscii     := ADR(stBmkAscii);
pstBmkAscii^[0] := STRING_TO_BYTE('');      // Pointer Cleaning Byte 0

IF pstBMK <> 0 AND pstBmkAscii <> 0 AND StBMK <> '' THEN
    //===========================================================================================================================================================================================================================================//
    //  BMK TO DINT Wandeln		                                                                          																															             //
    //===========================================================================================================================================================================================================================================// 
    FOR iFor := 0 TO LEN(stBMK) BY 1 DO
        iAkt    :=  BYTE_TO_INT(pstBMK^[iFor]);
        pstBmkAscii^[iFor + iOfset + 1] := STRING_TO_BYTE('');                                                          // Byte in Pointer Cleanen 
        IF BYTE_TO_INT(pstBMK^[iFor])>= 48 AND BYTE_TO_INT(pstBMK^[iFor]) <= 57 THEN                                    // ASCII Zahlen von 48 bis 57 = 0 bis 9
            pstBmkAscii^[iFor + iOfset] := pstBMK^[iFor];
        ELSIF BYTE_TO_INT(pstBMK^[iFor])>= 65 AND BYTE_TO_INT(pstBMK^[iFor]) <= 90 THEN                                 // ASCII Grosbuchstaben von 65 bis 90 = A bis Z
            pstBmkAscii^                := CONCAT(pstBmkAscii^,INT_TO_STRING(BYTE_TO_INT(pstBMK^[iFor])));
            iOfset                      := iOfset + 1;                                                                  // Zeichenversatz von + 1 je buchstaben 
        ELSIF BYTE_TO_INT(pstBMK^[iFor])>= 97 AND BYTE_TO_INT(pstBMK^[iFor]) <= 120 THEN                                // ASCII kleinbuchstaben von 97 bis 120 = a bis z 
            pstBmkAscii^                := CONCAT(pstBmkAscii^,INT_TO_STRING(BYTE_TO_INT(pstBMK^[iFor])-32));           // ASCII Nr - 32 wandelt klein- in Grossbuchstaben 
            iOfset                      := iOfset + 1;                                                                  // Zeichenversatz von + 1 je buchstaben 
        ELSIF BYTE_TO_INT(pstBMK^[iFor])= 45 THEN
            pstBmkAscii^[iFor + iOfset] := INT_TO_BYTE(43);     
        END_IF;
    END_FOR;
    //===========================================================================================================================================================================================================================================//
    //  Nr ergänzen 		                                                                          																															                 //
    //===========================================================================================================================================================================================================================================// 
    // Nr auf anzahl Stellen prüfen
    IF diNr >= 0 AND diNr <= 9 THEN
        IF xNoZero THEN
            stBmkAscii := CONCAT(stBMKAscii,DINT_TO_STRING(diNr));                                                      // Bei 1-Stelliger Zahl ohne 0 vorangesetzt
        ELSE
            stBmkAscii := CONCAT(stBMKAscii,CONCAT('0',DINT_TO_STRING(diNr)));                                          // Bei 1-Stelliger Zahl 0 voransetzen
        END_IF;    
    ELSIF diNr  >= 10 AND diNr <= 99 THEN
        stBmkAscii := CONCAT(stBMKAscii,DINT_TO_STRING(diNr));  
    ELSE
        IF enReportTypeIn = enReportType.Error THEN
            GVL_Report.fbReportVisu.proIdMissmatch := CONCAT(stBMK,CONCAT(' Error-ID not between 0-99 ID:',TO_STRING(diNr)));
        ELSIF enReportTypeIn = enReportType.Warning THEN
            GVL_Report.fbReportVisu.proIdMissmatch := CONCAT(stBMK,CONCAT(' Warning-ID not between 0-99 ID:',TO_STRING(diNr)));
        ELSIF enReportTypeIn = enReportType.Info THEN
            GVL_Report.fbReportVisu.proIdMissmatch := CONCAT(stBMK,CONCAT(' Info-ID not between 0-99 ID:',TO_STRING(diNr)));
        END_IF;    
    END_IF;
    //===========================================================================================================================================================================================================================================//
    //  Ausgabe DINT    		                                                                          																															             //
    //===========================================================================================================================================================================================================================================// 
    IF LEN(stBmkAscii) <= 12 THEN 
        fcBmkToId := TO_ULINT(stBMKAscii);
    ELSE 
        fcBmkToId := 0;
	END_IF
ELSE
    fcBmkToId   :=  TO_ULINT(diNr);    
END_IF;

END_FUNCTION

// 30 Program Organization Units/VIS/fbReportVisu
FUNCTION_BLOCK fbReportVisu 
VAR_INPUT
    ITF_BMK_IN                      :   ctaAppBmk.ITF_BMK;
END_VAR
VAR_OUTPUT
    xIsThereAnAktiveError           :   BOOL;
    xHandLokal                      :   BOOL;
END_VAR
VAR
	(* Multi Client Implementation *)
	diForClient						:	DINT;
	ayenVisuTableType               :   ARRAY[0..GlobalKonstant.VISU_MAX_NUMBER_OF_CLIENTS] OF enTableType; 
	ayOffset 						:	ARRAY[0..GlobalKonstant.VISU_MAX_NUMBER_OF_CLIENTS] OF INT;     
	ayOffsetOld						:	ARRAY[0..GlobalKonstant.VISU_MAX_NUMBER_OF_CLIENTS] OF INT;                                 
    ayItfReports                    :   ARRAY[0..GlobalKonstant.VISU_MAX_NUMBER_OF_CLIENTS] OF ARRAY[0..GlobalKonstant.iUpperSizeTable] OF ITF_REPORTOBJECT;
    ayShowReport                    :   ARRAY[0..GlobalKonstant.VISU_MAX_NUMBER_OF_CLIENTS] OF ARRAY[0..GlobalKonstant.iUpperSizeTable] OF BOOL;
    ayFilterError					:   ARRAY[0..GlobalKonstant.VISU_MAX_NUMBER_OF_CLIENTS] OF BOOL;
	ayFilterWarning					:   ARRAY[0..GlobalKonstant.VISU_MAX_NUMBER_OF_CLIENTS] OF BOOL;
	ayFilterInfo					:   ARRAY[0..GlobalKonstant.VISU_MAX_NUMBER_OF_CLIENTS] OF BOOL;
	ayusiFilter                     :   ARRAY[0..GlobalKonstant.VISU_MAX_NUMBER_OF_CLIENTS] OF USINT; 
	 
	(* Config *) 
	fbConfigFile                    :   CtaSysConfig.fbConfigFile;
    scPara                          :   scPara;
	
	(* Reports *)
    ayReporter                      :   ARRAY[1..1] OF fbReporter;
    xFernQuitt                      :   BOOL;
	
	(* Helper *)
    diFor                            :   DINT;
    ayReload                         :   ARRAY[0..GlobalKonstant.VISU_MAX_NUMBER_OF_CLIENTS] OF BOOL;
	ayWaitToReload					 :	 ARRAY[0..GlobalKonstant.VISU_MAX_NUMBER_OF_CLIENTS] OF INT;
    ayReloadExtern                   :   ARRAY[0..GlobalKonstant.VISU_MAX_NUMBER_OF_CLIENTS] OF BOOL;
    ayReloadIntern                   :   ARRAY[0..GlobalKonstant.VISU_MAX_NUMBER_OF_CLIENTS] OF BOOL;
    ayFirstLoadCsvDone               :   ARRAY[0..GlobalKonstant.VISU_MAX_NUMBER_OF_CLIENTS] OF BOOL;  
    ayFirstLoadPendingDone           :   ARRAY[0..GlobalKonstant.VISU_MAX_NUMBER_OF_CLIENTS] OF BOOL; 
    ayFilterErrorOld				 :   ARRAY[0..GlobalKonstant.VISU_MAX_NUMBER_OF_CLIENTS] OF BOOL;
	ayFilterWarningOld	 		     :   ARRAY[0..GlobalKonstant.VISU_MAX_NUMBER_OF_CLIENTS] OF BOOL;
	ayFilterInfoOld 				 :   ARRAY[0..GlobalKonstant.VISU_MAX_NUMBER_OF_CLIENTS] OF BOOL;
    
    stIdMissmatch                   :   STRING;
	aLogs 							: 	ARRAY[0..13] OF ST_MariaDbLog;
END_VAR

actConfigFile();
(* Offset Multiclient*)
FOR diForClient := LOWER_BOUND(ayOffset,1) TO UPPER_BOUND(ayOffset,1) DO
	IF NOT ayFirstLoadPendingDone[diForClient] THEN
		ayFilterError[diForClient]          := TRUE;
		ayFilterWarning[diForClient]        := TRUE;
		ayFilterInfo[diForClient]           := TRUE;
	END_IF;
	IF ayFilterError[diForClient] 	<> 	ayFilterErrorOld[diForClient]  OR       
		ayFilterWarning[diForClient]<>  ayFilterWarningOld[diForClient]  OR  
		ayFilterInfo[diForClient]   <>	ayFilterInfoOld[diForClient]     THEN 
			ayReloadIntern[diForClient] := TRUE;		
	END_IF;
	IF ayOffset[diForClient] <> ayOffsetOld[diForClient] THEN
		ayWaitToReload[diForClient] := 0;
	ELSIF ayOffset[diForClient] = ayOffsetOld[diForClient] OR ayReloadExtern[diForClient] OR ayReloadIntern[diForClient] THEN
		IF ayWaitToReload[diForClient] = 2 THEN
			ayReload[diForClient] 			:= TRUE;
			ayWaitToReload[diForClient] 	:= 3;
		ELSIF ayWaitToReload[diForClient] < 2 THEN
			ayWaitToReload[diForClient] := ayWaitToReload[diForClient] + 1;
		ELSIF ayWaitToReload[diForClient] >= 3 AND (ayReloadExtern[diForClient] OR ayReloadIntern[diForClient] ) THEN
			ayWaitToReload[diForClient] := 0;
			ayReloadExtern[diForClient] := FALSE;
			ayReloadIntern[diForClient] := FALSE;
		END_IF;
	END_IF;	
	ayOffsetOld[diForClient] := ayOffset[diForClient];

	IF ayenVisuTableType[diForClient] = enTableType.PENDING_REPORTS THEN
		(* Get Pending Reports *)
		loadPending(diForClient);   
		ayFirstLoadCsvDone[diForClient] := FALSE;  
	ELSIF ayenVisuTableType[diForClient] = enTableType.HISTORY_REPORTS THEN
		(* Get History CSV*)
		loadHistory(diForClient);    
		ayFirstLoadPendingDone[diForClient] := FALSE;
	END_IF;	
	ayFilterErrorOld[diForClient]          :=ayFilterError[diForClient];     
	ayFilterWarningOld[diForClient]        :=ayFilterWarning[diForClient];   
	ayFilterInfoOld[diForClient]           :=ayFilterInfo[diForClient];      
END_FOR;
  
actEWI();
xIsThereAnAktiveError := GVL_Report.fbReportObjectFactory.proIsThereAnAktiveError;
xHandLokal := GVL_Report.diCountHand <> 0;

METHOD metGetReport : ITF_REPORTOBJECT
VAR_INPUT
    iArrayPos   :   INT;
	iClientId	:	INT;
END_VAR
VAR
    xOk     :   BOOL;
END_VAR
metGetReport := 0;
IF iArrayPos >= 0 AND iArrayPos <= GlobalKonstant.iUpperSizeTable THEN
    IF __QUERYINTERFACE(ayItfReports[iClientId][iArrayPos],metGetReport) THEN
        xOk := TRUE;    
    END_IF;
END_IF;
END_METHOD

METHOD metGetShowReport : BOOL
VAR_INPUT
    iArrayPos   :   INT;
	iClientId	:	INT;
END_VAR
IF iArrayPos >= 0 AND iArrayPos <= GlobalKonstant.iUpperSizeTable THEN
    metGetShowReport := ayShowReport[iClientId][iArrayPos];
END_IF;
END_METHOD

ACTION actConfigFile:
(* PArameter *)
fbConfigFile();
scPara.fbxEnSafetyFernQuitt(_usiParaNr := 1,itfConfigFb:=fbConfigFile   ,_WertInit := TRUE);
scPara.fbuiMaxFernQuitt    (_usiParaNr := 2,itfConfigFb:=fbConfigFile   ,_WertInit := 5);
END_ACTION

PROPERTY proQuittExtern : BOOL
SET
IF proQuittExtern AND NOT xFernQuitt THEN
    IF scPara.fbxEnSafetyFernQuitt.proValue THEN
        IF ayReporter[1].proGetCounts < scPara.fbuiMaxFernQuitt.proValue THEN
            GVL_Report.fbReportObjectFactory.metQuittAllReports();
            xFernQuitt        := TRUE;
        END_IF;
    ELSE
        GVL_Report.fbReportObjectFactory.metQuittAllReports();
        xFernQuitt        := TRUE;
	END_IF;
ELSIF NOT proQuittExtern THEN
    xFernQuitt        := FALSE;
END_IF;
END_SET
END_PROPERTY

METHOD loadHistory
VAR_INPUT
	diClientId	:	DINT;
END_VAR
VAR
	scReportMetaData            :   scReportMetaData;
	diStartId					:	DINT;
	diMaxOffset					:	DINT;
	diOffset					:	DINT;
	
END_VAR
(* Get ItF CSV*)
IF NOT ayFirstLoadCsvDone[diForClient] OR ayReload[diForClient] THEN
    IF NOT ayFirstLoadCsvDone[diForClient] THEN
        ayOffset[diClientId] := 1;
	END_IF;
	
	diMaxOffset	:= TO_DINT(MaxOffset(diClientId));
	diOffset	:= TO_DINT(ayOffset[diClientId]);
	diStartId 	:= diMaxOffset - 14 - diOffset;
	diStartId   := MAX(diStartId,1);
	Fc_MariaDbLogRead(xExecute := TRUE ,aLogs := aLogs,dwStartId := TO_DWORD(diStartId) ,uiCount := 14);
		
		
    FOR diFor := 0 TO GlobalKonstant.iUpperSizeTable DO	
        IF __QUERYINTERFACE(GVL_Report.fbReportObjectFactory.metCsvGetItf(diFor,diClientId),ayItfReports[diClientId][diFor]) THEN
            ayItfReports[diClientId][diFor].metDestroy();
			IF aLogs[diFor].id > 0 THEN
				(* Data Sync *)
				scReportMetaData.xActive					:= aLogs[diFor].stateActive;
				scReportMetaData.xIsQuitt					:= aLogs[diFor].isQuitt;
				scReportMetaData.xReportIn					:= aLogs[diFor].reportIn;
				scReportMetaData.xQuitt						:= FALSE;
				scReportMetaData.usiPrio					:= aLogs[diFor].prio;
				scReportMetaData.dtFrom						:= aLogs[diFor].dtFrom;
				scReportMetaData.dtTo						:= aLogs[diFor].dtTo;
				scReportMetaData.dwWritePosInCsv			:= TO_DWORD(aLogs[diFor].id);
				scReportMetaData.enReportacknowledgeType	:= aLogs[diFor].reportAcknowledgType;
				scReportMetaData.enReportType				:= aLogs[diFor].reportType;
				scReportMetaData.stAdditionalText			:= aLogs[diFor].additionalText;
				scReportMetaData.stReporterObjId			:= aLogs[diFor].objectId;
				scReportMetaData.stReportTextList			:= aLogs[diFor].reportTextList;
				scReportMetaData.stReportTxtId				:= aLogs[diFor].reportTextId;
				scReportMetaData.uliReportId				:= aLogs[diFor].reportId;				
				ayItfReports[diClientId][diFor].proSetMetaData := scReportMetaData;
				ayItfReports[diClientId][diFor].proReporterObjectId := aLogs[diFor].objectId;
				ayItfReports[diClientId][diFor].proSetInstancePath := aLogs[diFor].instancePath;
				ayShowReport[diClientId][diFor] := TRUE; 
            ELSE
                ayShowReport[diClientId][diFor] := FALSE; 
            END_IF;      
        END_IF;
        IF diFor = GlobalKonstant.iUpperSizeTable THEN
            ayFirstLoadCsvDone[diForClient] := TRUE;
        END_IF;        
    END_FOR;
	ayReload[diForClient] 			:= FALSE;
END_IF;
END_METHOD

ACTION actEWI:
(* Externe Quittierung *)
ayReporter[1].metReport(xSetReportIn                := xFernQuitt,
                        iReportID                   := 99,
                        enReportTypeIn              := enReportType.Warning,
                        enReportAcknowledgeTypeIn   := SEL(scPara.fbxEnSafetyFernQuitt.proValue,enReportacknowledgeType.Auto,enReportacknowledgeType.RetryN),
                        tDelay                      := T#0S,
                        ITF_BMK_IN                  := ITF_BMK_IN,
                        pstReportTextListIn         := ADR(GlobalKonstant.stTextListWarning),
                        stOptionalReportText        := CONCAT(' ',TO_STRING(TO_INT(scPara.fbuiMaxFernQuitt.proValue)-(ayReporter[1].proGetCounts + 1))),
                        iRetryTilReportLock         := TO_INT(scPara.fbuiMaxFernQuitt.proValue),
                        xResetCount                 := FALSE,
                        tReset                      := T#1D);
END_ACTION

//FB_Init ist immer implizit verfügbar und wird primär für die Initialisierung verwendet.
//Der Rückgabewert wird nicht ausgewertet. Für gezielte Einflussnahme können Sie
//die Methoden explizit deklarieren und darin mit dem Standard-Initialisierungscode 
//zusätzlichen Code bereitstellen. Sie können den Rückgabewert auswerten.
METHOD FB_Init: BOOL
VAR_INPUT    
bInitRetains: BOOL; // TRUE: Die Retain-Variablen werden initialisiert (Reset warm / Reset kalt)    
bInCopyCode: BOOL;  // TRUE: Die Instanz wird danach in den Kopiercode kopiert (Online-Change)
END_VAR
END_METHOD

METHOD metReload : BOOL
VAR_INPUT
END_VAR
VAR
	diForTemp : DINT;
END_VAR
FOR diForTemp := LOWER_BOUND(ayReloadExtern,1) TO UPPER_BOUND(ayReloadExtern,1) DO
	ayReloadExtern[diForTemp] := TRUE;
END_FOR;
END_METHOD

METHOD FilterWarning 
VAR_INPUT
	xFilterWarning	: 	BOOL;
	diClientId		:	DINT;
END_VAR
IF diClientId >= LOWER_BOUND(ayFilterWarning,1) AND diClientId <= UPPER_BOUND(ayFilterWarning,1) THEN
	ayFilterWarning[diClientId] := xFilterWarning;
	ayReloadIntern[diForClient] := TRUE;
	ayOffset[diClientId] := 0;
END_IF;
END_METHOD

METHOD SetFilterId
VAR_INPUT
	diClientId	:	DINT;
END_VAR
(* FILTER *) 
(* No Filter *)
IF ayFilterError[diClientId] AND ayFilterWarning[diClientId] AND ayFilterInfo[diClientId] THEN
	ayusiFilter[diClientId] := 0;
(* Only Error *)
ELSIF ayFilterError[diClientId] AND NOT ayFilterWarning[diClientId] AND NOT ayFilterInfo[diClientId] THEN
	ayusiFilter[diClientId] := 1;
(* Only Warning *)    
ELSIF NOT ayFilterError[diClientId] AND ayFilterWarning[diClientId] AND NOT ayFilterInfo[diClientId] THEN
	ayusiFilter[diClientId] := 2;
(* Only Info *)  
ELSIF NOT ayFilterError[diClientId] AND NOT ayFilterWarning[diClientId] AND ayFilterInfo[diClientId] THEN
	ayusiFilter[diClientId] := 3;    
(* Error and Warning*)  
ELSIF ayFilterError[diClientId] AND ayFilterWarning[diClientId] AND NOT ayFilterInfo[diClientId] THEN
	ayusiFilter[diClientId] := 4;        
(* Error and Info*)  
ELSIF ayFilterError[diClientId] AND NOT ayFilterWarning[diClientId] AND ayFilterInfo[diClientId] THEN
	ayusiFilter[diClientId] := 5;     
(* Warning and Info*)  
ELSIF NOT ayFilterError[diClientId] AND ayFilterWarning[diClientId] AND ayFilterInfo[diClientId] THEN
	ayusiFilter[diClientId] := 6;   
ELSE
	ayusiFilter[diClientId] := 0;
END_IF;
END_METHOD

METHOD loadPending
VAR_INPUT
	diClientId	:	DINT;
END_VAR
(* Get pending Reports *)
IF NOT ayFirstLoadPendingDone[diForClient] OR ayReload[diForClient] THEN
SetFilterId(diClientId);
GVL_Report.fbSort.metFilterCustom(ayusiFilter[diClientId],diClientID);
    IF NOT ayFirstLoadPendingDone[diForClient] THEN
        ayOffset[diClientId]:= 0;
	END_IF;
    FOR diFor := 0 TO GlobalKonstant.iUpperSizeTable DO
        IF 1 + ayOffset[diClientId] + diFor <= Parameter.diMaxObject THEN
            IF __QUERYINTERFACE(GVL_Report.ayItfSortetReportsCustom[diClientId][1 + ayOffset[diClientId] + diFor],ayItfReports[diClientId][diFor]) THEN // Array Custom starts by 1 
                IF ayItfReports[diClientId][diFor] <> 0 THEN   
                    ayShowReport[diClientId][diFor] := TRUE;   
                ELSE
                    ayShowReport[diClientId][diFor] := FALSE; 
                END_IF;      
            END_IF;
            IF diFor = GlobalKonstant.iUpperSizeTable THEN
                ayFirstLoadPendingDone[diForClient] := TRUE;
            END_IF; 
        END_IF;     
    END_FOR;
	ayReload[diForClient] 			:= FALSE;
END_IF;
END_METHOD

METHOD FilterInfo
VAR_INPUT
	xFilterInfo	: 	BOOL;
	diClientId		:	DINT;
END_VAR
VAR
	diForTemp	:	DINT;
END_VAR
IF diClientId >= LOWER_BOUND(ayFilterInfo,1) AND diClientId <= UPPER_BOUND(ayFilterInfo,1) THEN
	ayFilterInfo[diClientId] := xFilterInfo;
	ayReloadIntern[diForClient] := TRUE;
	ayOffset[diClientId] := 0;
END_IF;
END_METHOD

METHOD FilterError
VAR_INPUT
	xFilterError: 	BOOL;
	diClientId	:	DINT;
END_VAR
IF diClientId >= LOWER_BOUND(ayFilterError,1) AND diClientId <= UPPER_BOUND(ayFilterError,1) THEN
	ayFilterError[diClientId] := xFilterError;
	ayReloadIntern[diForClient] := TRUE;
	ayOffset[diClientId] := 0;
END_IF;
END_METHOD

PROPERTY proAnzReportsInTable : UINT
GET
proAnzReportsInTable := GVL_Report.fbSort.proAnzReportsInTable;
END_GET
END_PROPERTY

PROPERTY proIdMissmatch : STRING
SET
stIdMissmatch := proIdMissmatch;
END_SET
GET
proIdMissmatch := stIdMissmatch;
END_GET
END_PROPERTY

METHOD MaxOffset : UDINT
VAR_INPUT
	diClientId	:	DINT;
END_VAR
VAR
	udiMaxOffset : UDINT;
END_VAR
IF ayenVisuTableType[diClientId] = enTableType.PENDING_REPORTS THEN
    udiMaxOffset := LIMIT(0,TO_UDINT(proAnzReportsInTable),16#FFFFFFFF);
ELSIF ayenVisuTableType[diClientId] = enTableType.HISTORY_REPORTS THEN
    udiMaxOffset := GVL_Report.fbDataHandler.proGetCountsOfReports;
END_IF
MaxOffset := udiMaxOffset;
END_METHOD

END_FUNCTION_BLOCK

// 30 Program Organization Units/SQL/Fc_MariaDbLogRead
FUNCTION Fc_MariaDbLogRead : BOOL
VAR_INPUT
    xExecute    : BOOL;
    dwStartId   : DWORD;
    uiCount     : USINT;
END_VAR

VAR_IN_OUT
    aLogs : ARRAY[0..13] OF ST_MariaDbLog;
END_VAR

VAR_OUTPUT
    xBusy       : BOOL;
    xDone       : BOOL;
    xError      : BOOL;
    dwResult    : DWORD;
    uiCountRead : USINT;
END_VAR

VAR
    sCommand    : STRING(4095);
    sSQL        : STRING(4095);
    sStdOut     : STRING(8185);
    sTemp       : STRING(4095);

    Result      : RTS_IEC_RESULT;
    diStdOutLen : DINT;

    xExecuteOld : BOOL;

    i           : INT;
    j           : INT;

    sRow        : STRING(4095);
    sField      : STRING(512);
    sRemaining  : STRING(8185);

    iPos        : INT;
    iField      : INT;

    dwId        : DWORD;
    uiRead      : USINT;

    xRunning    : BOOL;

    // Trennzeichen
    cFieldSep   : STRING(1) := '|';
    cRowSep     : STRING(1) := '$$';
	cLF			: STRING(2) := '$N';

END_VAR

// =====================================================
// AUSGÄNGE ZURÜCKSETZEN
// =====================================================

xDone       := FALSE;
xError      := FALSE;
dwResult    := 0;
uiCountRead := 0;


// =====================================================
// FLANKE ERKENNEN
// =====================================================

IF xExecute AND NOT xExecuteOld THEN

    // -------------------------------------------------
    // Werte prüfen
    // -------------------------------------------------
	dwStartId := MAX(1,dwStartId);
	
    IF uiCount > 14 THEN
        uiCount := 14;
    END_IF;

    IF uiCount = 0 THEN
        xError := TRUE;
        xBusy := FALSE;
        dwResult := 1;
        RETURN;
    END_IF;


    // -------------------------------------------------
    // ARRAY LEEREN
    // -------------------------------------------------

    FOR i := 0 TO 13 DO

        aLogs[i].id                   := 0;
        aLogs[i].createdAt            := DT#1970-01-01-00:00:00;
        aLogs[i].reportType           := enReportType.Info;
        aLogs[i].reportId             := 0;
        aLogs[i].reporterText         := '';
        aLogs[i].reportText           := '';
        aLogs[i].dtFrom               := DT#1970-01-01-00:00:00;
        aLogs[i].dtTo                 := DT#1970-01-01-00:00:00;
        aLogs[i].isQuitt              := FALSE;
        aLogs[i].reportTextList       := '';
        aLogs[i].reportTextId         := '';
        aLogs[i].reportAcknowledgType := 0;
        aLogs[i].objectId             := '';
        aLogs[i].instancePath         := '';
        aLogs[i].additionalText       := '';
        aLogs[i].prio                 := 0;
        aLogs[i].reportIn             := FALSE;
        aLogs[i].stateActive          := FALSE;

    END_FOR;


    // =================================================
    // SQL AUFBAUEN
    // =================================================

    sSQL := '';

    sTemp := 'USE CtaMariaDb; ';

    StrConcatA(
        ADR(sTemp),
        ADR(sSQL),
        TO_INT(SIZEOF(sSQL))
    );


    // -------------------------------------------------
    // SELECT
    // -------------------------------------------------

    sTemp := 'SELECT CONCAT( ';

    StrConcatA(
        ADR(sTemp),
        ADR(sSQL),
        TO_INT(SIZEOF(sSQL))
    );


    // -------------------------------------------------
    // ID
    // -------------------------------------------------

    sTemp := 'id';

    StrConcatA(
        ADR(sTemp),
        ADR(sSQL),
        TO_INT(SIZEOF(sSQL))
    );

    sTemp := ',CHAR(9),';

    StrConcatA(
        ADR(sTemp),
        ADR(sSQL),
        TO_INT(SIZEOF(sSQL))
    );


    // -------------------------------------------------
    // CREATED_AT
    // -------------------------------------------------

    sTemp := 'DATE_FORMAT(created_at,$'%Y-%m-%d %H:%i:%s$')';

    StrConcatA(
        ADR(sTemp),
        ADR(sSQL),
        TO_INT(SIZEOF(sSQL))
    );

    sTemp := ',CHAR(9),';

    StrConcatA(
        ADR(sTemp),
        ADR(sSQL),
        TO_INT(SIZEOF(sSQL))
    );


    // -------------------------------------------------
    // EVENT TYPE
    // -------------------------------------------------

    sTemp := 'event_type';

    StrConcatA(
        ADR(sTemp),
        ADR(sSQL),
        TO_INT(SIZEOF(sSQL))
    );

    sTemp := ',CHAR(9),';

    StrConcatA(
        ADR(sTemp),
        ADR(sSQL),
        TO_INT(SIZEOF(sSQL))
    );


    // -------------------------------------------------
    // EVENT ID
    // -------------------------------------------------

    sTemp := 'event_id';

    StrConcatA(
        ADR(sTemp),
        ADR(sSQL),
        TO_INT(SIZEOF(sSQL))
    );

    sTemp := ',CHAR(9),';

    StrConcatA(
        ADR(sTemp),
        ADR(sSQL),
        TO_INT(SIZEOF(sSQL))
    );


    // -------------------------------------------------
    // OBJECT NAME
    // -------------------------------------------------

    sTemp := 'REPLACE(REPLACE(IFNULL(object_name,$'$'),$'|$',$'/$'),$'$$$',$' $')';

    StrConcatA(
        ADR(sTemp),
        ADR(sSQL),
        TO_INT(SIZEOF(sSQL))
    );

    sTemp := ',CHAR(9),';

    StrConcatA(
        ADR(sTemp),
        ADR(sSQL),
        TO_INT(SIZEOF(sSQL))
    );


    // -------------------------------------------------
    // REPORTTEXT
    // -------------------------------------------------

    sTemp := 'REPLACE(REPLACE(IFNULL(reporttext,$'$'),$'|$',$'/$'),$'$$$',$' $')';

    StrConcatA(
        ADR(sTemp),
        ADR(sSQL),
        TO_INT(SIZEOF(sSQL))
    );

    sTemp := ',CHAR(9),';

    StrConcatA(
        ADR(sTemp),
        ADR(sSQL),
        TO_INT(SIZEOF(sSQL))
    );


    // -------------------------------------------------
    // DT FROM
    // -------------------------------------------------

    sTemp := 'IFNULL(DATE_FORMAT(dt_from,$'%Y-%m-%d %H:%i:%s$'),$'$')';

    StrConcatA(
        ADR(sTemp),
        ADR(sSQL),
        TO_INT(SIZEOF(sSQL))
    );

    sTemp := ',CHAR(9),';

    StrConcatA(
        ADR(sTemp),
        ADR(sSQL),
        TO_INT(SIZEOF(sSQL))
    );


    // -------------------------------------------------
    // DT TO
    // -------------------------------------------------

    sTemp := 'IFNULL(DATE_FORMAT(dt_to,$'%Y-%m-%d %H:%i:%s$'),$'$')';

    StrConcatA(
        ADR(sTemp),
        ADR(sSQL),
        TO_INT(SIZEOF(sSQL))
    );

    sTemp := ',CHAR(9),';

    StrConcatA(
        ADR(sTemp),
        ADR(sSQL),
        TO_INT(SIZEOF(sSQL))
    );


    // -------------------------------------------------
    // IS QUITT
    // -------------------------------------------------

    sTemp := 'IF(is_quitt,1,0)';

    StrConcatA(
        ADR(sTemp),
        ADR(sSQL),
        TO_INT(SIZEOF(sSQL))
    );

    sTemp := ',CHAR(9),';

    StrConcatA(
        ADR(sTemp),
        ADR(sSQL),
        TO_INT(SIZEOF(sSQL))
    );


    // -------------------------------------------------
    // REPORT TEXT LIST
    // -------------------------------------------------

    sTemp := 'REPLACE(REPLACE(IFNULL(report_textlist,$'$'),$'|$',$'/$'),$'$$$',$' $')';

    StrConcatA(
        ADR(sTemp),
        ADR(sSQL),
        TO_INT(SIZEOF(sSQL))
    );

    sTemp := ',CHAR(9),';

    StrConcatA(
        ADR(sTemp),
        ADR(sSQL),
        TO_INT(SIZEOF(sSQL))
    );


    // -------------------------------------------------
    // TEXT ID
    // -------------------------------------------------

    sTemp := 'IFNULL(text_id,0)';

    StrConcatA(
        ADR(sTemp),
        ADR(sSQL),
        TO_INT(SIZEOF(sSQL))
    );

    sTemp := ',CHAR(9),';

    StrConcatA(
        ADR(sTemp),
        ADR(sSQL),
        TO_INT(SIZEOF(sSQL))
    );


    // -------------------------------------------------
    // ACKNOWLEDGEMENT TYPE
    // -------------------------------------------------

    sTemp := 'IFNULL(type_acknowledg,0)';

    StrConcatA(
        ADR(sTemp),
        ADR(sSQL),
        TO_INT(SIZEOF(sSQL))
    );

    sTemp := ',CHAR(9),';

    StrConcatA(
        ADR(sTemp),
        ADR(sSQL),
        TO_INT(SIZEOF(sSQL))
    );


    // -------------------------------------------------
    // OBJECT ID
    // -------------------------------------------------

    sTemp := 'REPLACE(REPLACE(IFNULL(object_id,$'$'),$'|$',$'/$'),$'$$$',$' $')';

    StrConcatA(
        ADR(sTemp),
        ADR(sSQL),
        TO_INT(SIZEOF(sSQL))
    );

    sTemp := ',CHAR(9),';

    StrConcatA(
        ADR(sTemp),
        ADR(sSQL),
        TO_INT(SIZEOF(sSQL))
    );


    // -------------------------------------------------
    // INSTANCE PATH
    // -------------------------------------------------

    sTemp := 'REPLACE(REPLACE(IFNULL(instance_path,$'$'),$'|$',$'/$'),$'$$$',$' $')';

    StrConcatA(
        ADR(sTemp),
        ADR(sSQL),
        TO_INT(SIZEOF(sSQL))
    );

    sTemp := ',CHAR(9),';

    StrConcatA(
        ADR(sTemp),
        ADR(sSQL),
        TO_INT(SIZEOF(sSQL))
    );


    // -------------------------------------------------
    // ADDITIONAL TEXT
    // -------------------------------------------------

    sTemp := 'REPLACE(REPLACE(IFNULL(additional_text,$'$'),$'|$',$'/$'),$'$$$',$' $')';

    StrConcatA(
        ADR(sTemp),
        ADR(sSQL),
        TO_INT(SIZEOF(sSQL))
    );

    sTemp := ',CHAR(9),';

    StrConcatA(
        ADR(sTemp),
        ADR(sSQL),
        TO_INT(SIZEOF(sSQL))
    );


    // -------------------------------------------------
    // PRIO
    // -------------------------------------------------

    sTemp := 'IFNULL(prio,0)';

    StrConcatA(
        ADR(sTemp),
        ADR(sSQL),
        TO_INT(SIZEOF(sSQL))
    );

    sTemp := ',CHAR(9),';

    StrConcatA(
        ADR(sTemp),
        ADR(sSQL),
        TO_INT(SIZEOF(sSQL))
    );


    // -------------------------------------------------
    // IN STATE
    // -------------------------------------------------

    sTemp := 'IF(in_state,1,0)';

    StrConcatA(
        ADR(sTemp),
        ADR(sSQL),
        TO_INT(SIZEOF(sSQL))
    );

    sTemp := ',CHAR(9),';

    StrConcatA(
        ADR(sTemp),
        ADR(sSQL),
        TO_INT(SIZEOF(sSQL))
    );


    // -------------------------------------------------
    // STATE
    // -------------------------------------------------

    sTemp := 'IF(state,1,0))';

    StrConcatA(
        ADR(sTemp),
        ADR(sSQL),
        TO_INT(SIZEOF(sSQL))
    );


    // =================================================
    // WHERE
    // =================================================

    sTemp := ' FROM logs WHERE id BETWEEN ';

    StrConcatA(
        ADR(sTemp),
        ADR(sSQL),
        TO_INT(SIZEOF(sSQL))
    );

    sTemp := DWORD_TO_STRING(dwStartId);

    StrConcatA(
        ADR(sTemp),
        ADR(sSQL),
        TO_INT(SIZEOF(sSQL))
    );

    sTemp := ' AND ';

    StrConcatA(
        ADR(sTemp),
        ADR(sSQL),
        TO_INT(SIZEOF(sSQL))
    );


	sTemp := UDINT_TO_STRING(TO_UDINT(dwStartId) + TO_UDINT(uiCount));
	 
    StrConcatA(
        ADR(sTemp),
        ADR(sSQL),
        TO_INT(SIZEOF(sSQL))
    );

    // =================================================
    // ORDER
    // =================================================

    sTemp := ' ORDER BY id DESC;';

    StrConcatA(
        ADR(sTemp),
        ADR(sSQL),
        TO_INT(SIZEOF(sSQL))
    );

   

    // =================================================
    // MARIADB COMMAND
    // =================================================

    sCommand := '';

    sTemp :=
        'mariadb --socket=/var/lib/mysql/mysql.sock ';

    StrConcatA(
        ADR(sTemp),
        ADR(sCommand),
        TO_INT(SIZEOF(sCommand))
    );


    sTemp :=
        '-u root -pCTA-MariaDb1981! ';

    StrConcatA(
        ADR(sTemp),
        ADR(sCommand),
        TO_INT(SIZEOF(sCommand))
    );


    sTemp :=
        '--default-character-set=utf8mb4 ';

    StrConcatA(
        ADR(sTemp),
        ADR(sCommand),
        TO_INT(SIZEOF(sCommand))
    );


    sTemp :=
        '-N -B -e "';

    StrConcatA(
        ADR(sTemp),
        ADR(sCommand),
        TO_INT(SIZEOF(sCommand))
    );


    // SQL anhängen

    StrConcatA(
        ADR(sSQL),
        ADR(sCommand),
        TO_INT(SIZEOF(sCommand))
    );


    sTemp := '"';

    StrConcatA(
        ADR(sTemp),
        ADR(sCommand),
        TO_INT(SIZEOF(sCommand))
    );


    // =================================================
    // SQL AUSFÜHREN
    // =================================================

    sStdOut := '';

